// TwinCAT 3 PLC project PLC1
// ProgramVersion: 3.1.4023.0
// libraries:
//   Tc2_EtherCAT, * (Beckhoff Automation GmbH)
//   Tc2_MC2, * (Beckhoff Automation GmbH)
//   Tc2_Standard, * (Beckhoff Automation GmbH)
//   Tc2_SUPS, * (Beckhoff Automation GmbH)
//   Tc2_System, * (Beckhoff Automation GmbH)
//   Tc2_Utilities, * (Beckhoff Automation GmbH)
//   Tc3_MC2_AdvancedHoming, * (Beckhoff Automation GmbH)
//   Tc3_Module, * (Beckhoff Automation GmbH)
//   VisuDialogs, * (System)
// project tree:
//   / GlobalTextList.TcGTLO, PlcTask.TcTTO, Visualization Manager.TcVMO (not stored)
//   GVLs/ GVL_APP.TcGVL
//   POUs/Application_Specific/Applications/ Application_Template.TcPOU
//   POUs/Application_Specific/Axes/ Axis_Template.TcPOU, Pneumatics_Template.TcPOU
//   POUs/ MAIN.TcPOU
//   tc_mca_std_lib/DUTs/Axis_Structures/ ST_AxisConfig.TcDUT, ST_AxisControl.TcDUT, ST_AxisDescription.TcDUT, ST_AxisError.TcDUT, ST_AxisInputs.TcDUT, ST_AxisPersistent.TcDUT, ST_AxisStatus.TcDUT, ST_AxisStruct.TcDUT, ST_GearAxis.TcDUT, ST_HomingConfig.TcDUT
//   tc_mca_std_lib/DUTs/ E_AxisEngUnit.TcDUT, E_AxisParameters.TcTLEO, E_HomingRoutines.TcTLEO, E_MonitoringLedFunction.TcDUT, E_MotionFunctions.TcDUT, E_RestorePosition.TcDUT, E_SlitPairStates.TcDUT, E_SlitPairStatesV2.TcDUT, I_Axis.TcIO, ST_McStatus.TcDUT, ST_MonitoringAlarm.TcDUT
//   tc_mca_std_lib/DUTs/Pneumatics/ E_PneumaticAxisErrors.TcDUT, E_PneumaticMode.TcDUT, ST_PneumaticAxisConfig.TcDUT, ST_PneumaticAxisControl.TcDUT, ST_PneumaticAxisError.TcDUT, ST_PneumaticAxisInputs.TcDUT, ST_PneumaticAxisOutputs.TcDUT, ST_PneumaticAxisStatus.TcDUT, ST_PneumaticAxisStruct.TcDUT
//   tc_mca_std_lib/GVLs/ GVL.TcGVL
//   tc_mca_std_lib/POUs/ FB_ESSMonitoring.TcPOU
//   tc_mca_std_lib/POUs/Motion/ FB_Axis.TcPOU, FB_SlitPair.TcPOU, FB_SlitPairV2.TcPOU
//   tc_mca_std_lib/POUs/Motion/Homing/ FB_Homing.TcPOU
//   tc_mca_std_lib/POUs/Pneumatics/ FB_PneumaticAxis.TcPOU
//   tc_mca_std_lib/VISUs/ languageSupport.TcTLO, MainVisu.TcVIS, ParameterTextList.TcTLO, PneumaticsVisu.TcVIS
//   tc_mca_std_lib/VISUs_Org/ languageSupport_1.TcTLO, MainVisu_1.TcVIS, ParameterTextList_1.TcTLO, PneumaticsVisu_1.TcVIS
// real-time tasks:
//   TASK PlcTask: cycle T#10ms, priority 20, ADS port 350
// motion (NC):
//   TASK NC-Task 1 SAF: cycle T#2ms, priority 4, ADS port 501
//   TASK NC-Task 1 SVB: cycle T#10ms, priority 8, ADS port 511
//   AXIS Axis 1_X1 (id 1)
//     OtherSettings: AllowMotionCmdToSlave=true
//     encoder EncType=1
//     drive DrvType=5
//       Analog: TorqueSetpointScale=10, ScaleFactorActTorque=0.1
//       TimeComp: TaskDelayCycles=1
//     controller CtrType=1
//       CtrPara: PriorControlFactor=1
//         Observer: BandWidth=20
//   AXIS Axis 2_Y (id 2)
//     OtherSettings: AllowMotionCmdToSlave=true
//     encoder EncType=1
//     drive DrvType=5
//       Analog: TorqueSetpointScale=10, ScaleFactorActTorque=0.1
//       TimeComp: TaskDelayCycles=1
//     controller CtrType=1
//       CtrPara: PriorControlFactor=1
//         Observer: BandWidth=20
//   AXIS Axis 3_Z (id 3)
//     OtherSettings: AllowMotionCmdToSlave=true
//     encoder EncType=1
//     drive DrvType=5
//       Analog: TorqueSetpointScale=10, ScaleFactorActTorque=0.1
//       TimeComp: TaskDelayCycles=1
//     controller CtrType=1
//       CtrPara: PriorControlFactor=1
//         Observer: BandWidth=20
//   AXIS Axis 4_X2 (id 4)
//     OtherSettings: AllowMotionCmdToSlave=true
//     encoder EncType=1
//     drive DrvType=5
//       Analog: TorqueSetpointScale=10, ScaleFactorActTorque=0.1
//       TimeComp: TaskDelayCycles=1
//     controller CtrType=1
//       CtrPara: PriorControlFactor=1
//         Observer: BandWidth=20
// variable links:
//   PLC1/PLC1 Instance <-> NC-Task 1 SAF/Axes/Axis 1_X1
//     PlcTask Inputs/GVL.astAxes[1].Axis.NcToPlc <-> Outputs/ToPlc
//     PlcTask Outputs/GVL.astAxes[1].Axis.PlcToNc <-> Inputs/FromPlc
//   PLC1/PLC1 Instance <-> NC-Task 1 SAF/Axes/Axis 2_Y
//     PlcTask Inputs/GVL.astAxes[2].Axis.NcToPlc <-> Outputs/ToPlc
//     PlcTask Outputs/GVL.astAxes[2].Axis.PlcToNc <-> Inputs/FromPlc
//   PLC1/PLC1 Instance <-> NC-Task 1 SAF/Axes/Axis 3_Z
//     PlcTask Inputs/GVL.astAxes[3].Axis.NcToPlc <-> Outputs/ToPlc
//     PlcTask Outputs/GVL.astAxes[3].Axis.PlcToNc <-> Inputs/FromPlc
//   PLC1/PLC1 Instance <-> NC-Task 1 SAF/Axes/Axis 4_X2
//     PlcTask Inputs/GVL.astAxes[4].Axis.NcToPlc <-> Outputs/ToPlc
//     PlcTask Outputs/GVL.astAxes[4].Axis.PlcToNc <-> Inputs/FromPlc

CONFIGURATION PLC1
    RESOURCE PLC ON TwinCAT3
        TASK PlcTask(INTERVAL := T#10ms, PRIORITY := 20);
        PROGRAM MAIN WITH PlcTask : MAIN;
    END_RESOURCE
END_CONFIGURATION

// ---- tc_mca_std_lib/DUTs/Axis_Structures/ST_AxisConfig.TcDUT
(*These are axis parameters that are set up during commissioning and
in theory don't neeed to be change as part of daily moving of axes.
For instance they may be changed due to poor parameter selection
or change of instrument configuration.*)
TYPE ST_AxisConfig :
STRUCT
    //Axis Parameters
    fOverride: LREAL := 100; //Controller override %, used a global scale for an axis in terms of velocity. Generally set to 100%.
    fHomePosition: LREAL := 0; //The position that the axis should be set to once homing is completed
    fHomeFinishDistance: LREAL := 0; //Distrance that the axis should move back into the working zone after homing is finished
    eHomeSeq: E_HomingRoutines; //Homing sequence to perform
    eRestorePosition: E_RestorePosition; //Restore position of incremental axis after loss of power to the CPU, 0=don't restore, 1=restore but don't home

    //Advanced homing parameters
    stHomingConfig: ST_HomingConfig; //Structure containing the advanced homing parameters

    //Temperature disable configuration
    bEnableTemperatureDisable: BOOL := FALSE; //Enable disabling axis because of high temperature
    fMaxTemperature: LREAL := 0.0;
    fTempScalingFactor: REAL := 10.0;

    //Read and Write parameters
    eAxisParameters: E_AxisParameters; //Enumeration of axis parameters
    fWriteAxisParameter: LREAL; //The value to be writen to eAxisParameterNumber
    fReadAxisParameter: LREAL; //Read the current value of the selected eAxisParameterNumber

    //Multi master axis parameters
    astMultiMasterAxis: ARRAY [1..4] OF ST_GearAxis;
    astMultiMasterAxisLatched: ARRAY [1..4] OF ST_GearAxis; //A kind of readback since one doesn't exist in AXIS_REF
    afMultiSlaveAxisRatio: ARRAY [1..GVL_APP.nAXIS_NUM] OF LREAL;

    // Read only MC parameters
    bReadMcParametersValid: BOOL:= FALSE;
    bReadMcParametersError: BOOL:= FALSE;
    fVelocityDefaultSlow: LREAL; //Read only - AxisVeloManSlow
    fVelocityDefaultFast: LREAL; //Read only - AxisVeloManFast
    fHomingVelToCam: LREAL; //Read only - AxisCalibrationVelocityForward
    fHomingVelFromCam: LREAL; //Read only - AxisCalibrationVelocityBackward
    fVeloMax: LREAL; //Read only - AxisMaxVelocity
    fMaxAcc: LREAL; //Read only - AxisMaximumAcceleration
    fMaxDec: LREAL; //Read only - AxisMaxDeceleration
    fDefaultAcc: LREAL; //Read only - AxisDefaultAcceleration
    fDefaultDec: LREAL; //Read only - AxisDefaultDeceleration
    bEnMinSoftPosLimit: BOOL; //Read only
    fMinSoftPosLimit: LREAL; //Read only
    bEnMaxSoftPosLimit: BOOL; //Read only
    fMaxSoftPosLimit: LREAL; //Read only
    bEnPositionLagMonitoring: BOOL; //Read only
    fMaxPosLagValue: LREAL; //Read only
    bEnTargetPositionMonitoring: BOOL; //Read only
    fTargetPositionWindow: LREAL; //Read only
END_STRUCT
END_TYPE

// ---- tc_mca_std_lib/DUTs/Axis_Structures/ST_AxisControl.TcDUT
(*These are parameters that are used to initiate axis movements
They are commands that are commonly used commands*)
TYPE ST_AxisControl :
STRUCT
    //Actions from controls system
    bExecute: BOOL; //Rising edge to execute some motion FB's
    bReset: BOOL; //Reset axis from Error state
    bStop: BOOL;
    bHalt: BOOL;
    bEnable: BOOL; //Enable axis drive
    bJogFwd: BOOL;
    bJogBwd: BOOL;
    bInterlockFwd: BOOL := FALSE; //Bit for interlocking motors in the positive direction
    bInterlockBwd: BOOL := FALSE; //Bit for interlocking motors in the negative direction
    eCommand: E_MotionFunctions;
    fVelocity: LREAL; //Velocity must be specified
    fJogVelocity: LREAL; //Jogging velocity
    fAcceleration: LREAL; //Not all FBs use, 0 is NC default
    fDeceleration: LREAL;
    fPosition: LREAL; //The position to move to for an absolute move and the amount to move in a relative move
    bHWMaskActive: BOOL := FALSE;
    fMaskedTemperature: LREAL := 0.0;
END_STRUCT
END_TYPE

// ---- tc_mca_std_lib/DUTs/Axis_Structures/ST_AxisDescription.TcDUT
TYPE ST_AxisDescription :
STRUCT
    sAxisName : STRING(nMAX_AXIS_NAME);
    eUnit: E_AxisEngUnit; //Code for the axis base unit (like m or degree)
    nPrefix: INT; //Exponent defining unit prefix, e.g. 3 for k(kilo)
END_STRUCT
END_TYPE

// ---- tc_mca_std_lib/DUTs/Axis_Structures/ST_AxisError.TcDUT
TYPE ST_AxisError:
STRUCT
//PLCopen function block errors
    nPowerErrorID: UDINT;
    nMoveAbsoluteErrorID: UDINT;
    nMoveRelativeErrorID: UDINT;
    nMoveVelocityErrorID: UDINT;
    nMoveModuloErrorID: UDINT;
    nHomeErrorID: UDINT;
    nHaltErrorID: UDINT;
    nResetErrorID: UDINT;
    nStopErrorID: UDINT;
    nGearInMultiMasterErrorID: UDINT;
    nGearOutErrorID: UDINT;
    nWriteParameterErrorId: UDINT;
    nReadParameterErrorId: UDINT;
//Error from the NC
    nNCErrorID : UDINT;
END_STRUCT
END_TYPE

// ---- tc_mca_std_lib/DUTs/Axis_Structures/ST_AxisInputs.TcDUT
TYPE ST_AxisInputs :
STRUCT
    bLimitFwd AT %I*: BOOL;
    bLimitBwd AT %I*: BOOL;
    bHomeSensor AT %I*: BOOL; //Reference siganl for homing
    nTempPT100 AT %I*: INT;
END_STRUCT
END_TYPE

// ---- tc_mca_std_lib/DUTs/Axis_Structures/ST_AxisPersistent.TcDUT
TYPE ST_AxisPersistent :
STRUCT
    //Settings for restoring positions on power off
    fPositionAtShutdown: LREAL; //The position that the axis was at when CPU shut down
    fEncoderBiasAtShutdown: LREAL; //Encoder position BIAS value when CPU shut down
    bMovingAtShutdown: BOOL; //True if the axis was moving at shutdown, False otherwise
END_STRUCT
END_TYPE

// ---- tc_mca_std_lib/DUTs/Axis_Structures/ST_AxisStatus.TcDUT
TYPE ST_AxisStatus :
STRUCT
    //Outputs & Status
    bAxisInitialized: BOOL := FALSE; //True when all parameters from actReadMcParameters are valid
    bEnabled: BOOL; //Axis drive enabled
    bCommandAborted: BOOL; //Command aborted output of the eCommand function blocks
    bBusy: BOOL; //Axis busy (eCommand function block is active)
    bDone: BOOL; //Last eCommand function block executed successfully;
    //bDone will also be set with the InGear and InVelocity outputs
    //When InVelocity is set, fbMoveVelocity is still acitve, which is reflected by the bBusy status
    bInVelocity: BOOL; //MC_MoveVelocity has reached target velocity; will stay true until the movement stops
    bHomed: BOOL; //Axis homed
    bMoving: BOOL; //Moving state from the NC
    bMovingForward: BOOL; //Moving forward indicator from NC
    bMovingBackward: BOOL; //Moving backward indicator from NC
    bInTargetPosition: BOOL; //In target position bit from AxisStatus()
    bFwEnabled: BOOL; //Positive movement of axis is enabled/disabled
    bBwEnabled: BOOL; //Negative movement of axis is enabled/disabled
    bInterlockedFwd: BOOL; //Axis interlocked in the postive direction
    bInterlockedBwd: BOOL; //Axis interlocked in the negative direction
    bGeared: BOOL; //Axis is an active slave
    bCoupledGear1: BOOL;
    bCoupledGear2: BOOL;
    bCoupledGear3: BOOL;
    bCoupledGear4: BOOL;
    fActPosition: LREAL; //Actual position value
    fActTemperature: LREAL; //Actual Temperature
    bHighTempAxisDisabled: BOOL := FALSE; //Bit for disabling the axis when temperature too high
    nEncoderRawCounter AT %I*: UDINT; //Raw encoder counter value
    nStepperDriveCounter AT %I*: UDINT; //Raw internal counter from stepper drive
    fActVelocity: LREAL; //Actual velocity
    bError: BOOL; //Motion function block has produced error (NC drive not necessarily in error state)
    nErrorID: UDINT; //Last motion function block errorID or NC errorID
END_STRUCT
END_TYPE

// ---- tc_mca_std_lib/DUTs/Axis_Structures/ST_AxisStruct.TcDUT
TYPE ST_AxisStruct :
STRUCT
    stControl: ST_AxisControl;
    stStatus: ST_AxisStatus;
    stConfig: ST_AxisConfig;
    stError: ST_AxisError;
    stInputs: ST_AxisInputs;
    stDescription: ST_AxisDescription;
    //The NC axis link to the hardware that is controlling
    Axis: AXIS_REF;
END_STRUCT
END_TYPE

// ---- tc_mca_std_lib/DUTs/Axis_Structures/ST_GearAxis.TcDUT
TYPE ST_GearAxis :
STRUCT
    nIndex: UINT := 1; //Index of the master axis
    fRatio: LREAL := 0; //Gearing ratio between master axis and this one
END_STRUCT
END_TYPE

// ---- tc_mca_std_lib/DUTs/Axis_Structures/ST_HomingConfig.TcDUT
TYPE ST_HomingConfig :
STRUCT
    //Hardware signals
    eLimitSwitchMode: MC_Switch_Mode := mcRisingEdge;
    eRefSwitchMode: MC_Switch_Mode := mcRisingEdge;

    //General Advanced Homing Configuration
    bDisableDriveAccess: BOOL := TRUE; //Disables the drive access to drives. Standard for stepper motors. If supported in drive, can be set to FALSE, e.g. for AX5106.
    bEnableLagErrorDetection :BOOL := FALSE; // Keep the lag error detection active during homing
    bInstantLagReduction :BOOL := FALSE; //(belongs to Option4) When referencing to a mechanical fixed stop, it is purposeful in particular with "soft" fixed stops, the lag error is dissipated abruptly by setting this flag.
    tTimeLimit: TIME; // Exceeding this time leads to the search procedure being aborted.
    fDistanceLimit: LREAL; // Exceeding this distance in relation to the start position leads to the search procedure being aborted.
    fTorqueLimit: LREAL; // The motor torque is limited to this value, in relation to the weight counterbalance that is possibly parameterized in the drive, in order to avoid mechanical damage.

    //Homing Configuration for Step Block
    fDetectionVelocityLimit: LREAL; // Velocity that must be fallen below for the DetectionVelocityTime in order to detect driving against the fixed stop.
    tDetectionVelocityTime: TIME; // Time for detecting the velocity undershoot when driving against the fixed stop.
    fLagLimit: LREAL; // Position lag value which, if exceeded, leads to detection of driving against the fixed stop.
END_STRUCT
END_TYPE

// ---- tc_mca_std_lib/DUTs/E_AxisEngUnit.TcDUT
{attribute 'qualified_only'}
{attribute 'strict'}
TYPE E_AxisEngUnit :
(
    eMeter := 0,
    eDegree := 1
) := eMeter;
END_TYPE

// ---- tc_mca_std_lib/DUTs/E_AxisParameters.TcTLEO
{attribute 'qualified_only'}
{attribute 'strict'}
TYPE E_AxisParameters :
(
//PLCopen specific parameters Index-Group 0x4000 + ID
    CommandedPosition := 1, //lreal taken from NcToPlc
    SWLimitForward := 2, //lreal IndexOffset= 16#0001_000E
    SWLimitBackward := 3, //lreal IndexOffset= 16#0001_000D
    EnableLimitForward := 4, //bool IndexOffset= 16#0001_000C
    EnableLimitBackward := 5, //bool IndexOffset= 16#0001_000B
    EnablePositionLagMonitoring := 6, //bool IndexOffset= 16#0002_0010
    MaxPositionLag := 7, //lreal IndexOffset= 16#0002_0012
    AxisMaxVelocity := 8, //lreal IndexOffset= 16#0000_0027
    ActualVelocity := 10, //lreal taken from NcToPlc
    CommandedVelocity := 11, //lreal taken from NcToPlc
    AxisDefaultAcceleration := 12, //lreal IndexOffset= 16#0000_0101
    AxisDefaultDeceleration := 14, //lreal IndexOffset= 16#0000_0102
    AxisDefaultJerk := 16, //lreal IndexOffset= 16#0000_0103

//Beckhoff specific parameters Index-Group 0x4000 + ID
    AxisId := 1000, //lreal IndexOffset= 16#0000_0001
    AxisManualVelocitySlow := 1001, //lreal IndexOffset= 16#0000_0008
    AxisManualVelocityFast := 1002, //lreal IndexOffset= 16#0000_0009
    AxisRapidTraverseVelocity := 1009, //lreal IndexOffset= 16#0000_000A
    AxisVelocityToCam := 1012, //lreal IndexOffset= 16#0000_0006
    AxisVelocityFromCam := 1013, //lreal IndexOffset= 16#0000_0007
    AxisJogIncrementForward := 1014, //lreal IndexOffset= 16#0000_0018
    AxisJogIncrementBackward := 1015, //lreal IndexOffset= 16#0000_0019
    MaxPositionLagFilterTime := 1022, //lreal IndexOffset= 16#0002_0013
    AxisEnPositionRangeMonitoring := 1023, //bool IndexOffset= 16#0000_000F
    AxisPositionRangeWindow := 1024, //lreal IndexOffset= 16#0000_0010
    AxisEnTargetPositionMonitoring:= 1025, //bool IndexOffset= 16#0000_0015
    AxisTargetPositionWindow := 1026, //lreal IndexOffset= 16#0000_0016
    AxisTargetPositionMonitoringTime := 1027, //lreal IndexOffset= 16#0000_0017
    AxisEnInTargetTimeout := 1028, //bool IndexOffset= 16#0000_0029
    AxisInTargetTimeout := 1029, //lreal IndexOffset= 16#0000_002A
    AxisEnMotionMonitoring := 1030, //bool IndexOffset= 16#0000_0011
    AxisMotionMonitoringWindow := 1031, //lreal IndexOffset= 16#0000_0028
    AxisMotionMonitoringTime := 1032, //lreal IndexOffset= 16#0000_0012
    AxisDelayTimeVeloPosition := 1033, //lreal IndexOffset= 16#0000_0104
    AxisEnLoopingDistance := 1034, //bool IndexOffset= 16#0000_0013
    AxisLoopingDistance := 1035, //lreal IndexOffset= 16#0000_0014
    AxisEnBacklashCompensation := 1036, //bool IndexOffset= 16#0000_002B
    AxisBacklash := 1037, //lreal IndexOffset= 16#0000_002C
    AxisEnDataPersistence := 1038, //bool IndexOffset= 16#0000_0030
    AxisRefVeloOnRefOutput := 1039, //lreal IndexOffset= 16#0003_0101
    AxisOverrideType := 1040, //lreal IndexOffset= 16#0000_0105
    //new since 4/2007
    AxisEncoderOffset := 1042, //lreal IndexOffset= 16#0001_0007
    AxisEncoderDirectionInverse := 1043, //bool IndexOffset= 16#0001_0008
    AxisEncoderMask := 1044, //dword IndexOffset= 16#0001_0015
    AxisEncoderModuloValue := 1045, //lreal IndexOffset= 16#0001_0009
    AxisModuloToleranceWindow := 1046, //lreal IndexOffset= 16#0001_001B
    AxisEnablePosCorrection := 1047, //bool IndexOffset= 16#0001_0016
    AxisPosCorrectionFilterTime := 1048, //lreal IndexOffset= 16#0001_0017
    //new since 1/2010
    AxisUnitInterpretation := 1049, //lreal IndexOffset= 16#0000_0026
    AxisMotorDirectionInverse := 1050, //bool  IndexOffset= 16#0003_0006
    //new since 1/2011
    AxisCycleTime := 1051, //lreal IndexOffset= 16#0000_0004
    //new since 5/2011
    AxisFastStopSignalType := 1052, //dword IndexOffset= 16#0000_001E
    AxisFastAcc := 1053, //lreal IndexOffset= 16#0000_010A
    AxisFastDec := 1054, //lreal IndexOffset= 16#0000_010B
    AxisFastJerk := 1055, //lreal IndexOffset= 16#0000_010C
    // new since 1/2012 *)
    AxisEncoderScalingNumerator := 1056, //lreal IndexOffset= 16#0001_0023 - available in Tc3
    AxisEncoderScalingDenominator := 1057, //lreal IndexOffset= 16#0001_0024 - available in Tc3
    (* new since 7/2016 *)
    AxisMaximumAcceleration := 1058, //lreal IndexOffset= 16#0000_00F1
    AxisMaximumDeceleration := 1059, //lreal IndexOffset= 16#0000_00F2
    AxisVeloJumpFactor := 1060, //lreal IndexOffset= 16#0000_0106
    AxisToleranceBallAuxAxis := 1061, //lreal IndexOffset= 16#0000_0108
    AxisMaxPositionDeviationAuxAxis := 1062, //lreal IndexOffset= 16#0000_0109
    AxisErrorPropagationMode := 1063, //dword IndexOffset= 16#0000_001A
    AxisErrorPropagationDelay := 1064, //lreal IndexOffset= 16#0000_001B
    AxisCoupleSlaveToActualValues := 1065, //bool IndexOffset= 16#0000_001C
    AxisAllowMotionCmdToSlaveAxis := 1066, //bool IndexOffset= 16#0000_0020
    AxisAllowMotionCmdToExtSetAxis := 1067, //bool IndexOffset= 16#0000_0021
    AxisEncoderSubMask := 1068, //dword IndexOffset= 16#0001_0108
    AxisEncoderReferenceSystem := 1069, //dword IndexOffset= 16#0001_0019
    AxisEncoderPositionFilterPT1 := 1070, //lreal IndexOffset= 16#0001_0010
    AxisEncoderVelocityFilterPT1 := 1071, //lreal IndexOffset= 16#0001_0011
    AxisEncoderAccelerationFilterPT1 := 1072, //lreal IndexOffset= 16#0001_0012
    AxisEncoderMode := 1073, //dword IndexOffset= 16#0001_000A
    AxisEncoderHomingInvDirCamSearch := 1074, //bool IndexOffset= 16#0001_0101
    AxisEncoderHomingInvDirSyncSearch := 1075, //bool IndexOffset= 16#0001_0102
    AxisEncoderHomingCalibValue := 1076, //lreal IndexOffset= 16#0001_0103
    AxisEncoderReferenceMode := 1077, //dword IndexOffset= 16#0001_0107
    AxisRefVeloOutputRatio := 1078, //lreal IndexOffset= 16#0003_0102
    AxisDrivePositionOutputScaling := 1079, //lreal IndexOffset= 16#0003_0109
    AxisDriveVelocityOutputScaling := 1080, //lreal IndexOffset= 16#0003_0105
    AxisDriveVelocityOutputDelay := 1081, //lreal IndexOffset= 16#0003_010D
    AxisDriveMinOutputLimitation := 1082, //lreal IndexOffset= 16#0003_000B
    AxisDriveMaxOutputLimitation := 1083, //lreal IndexOffset= 16#0003_000C
    AxisTorqueInputScaling := 1084, //lreal IndexOffset= 16#0003_0031 - available in Tc3
    AxisTorqueInputFilterPT1 := 1085, //lreal IndexOffset= 16#0003_0032 - available in Tc3
    AxisTorqueDerivationInputFilterPT1 := 1086, //lreal IndexOffset= 16#0003_0033 - available in Tc3
    AxisTorqueOutputScaling := 1087, //lreal IndexOffset= 16#0003_010B
    AxisTorqueOutputDelay := 1088, //lreal IndexOffset= 16#0003_010F
    AxisAccelerationOutputScaling := 1089, //lreal IndexOffset= 16#0003_010A
    AxisAccelerationOutputDelay := 1090, //lreal IndexOffset= 16#0003_010E
    AxisDrivePositionOutputSmoothFilterType := 1091, //dword IndexOffset= 16#0003_0110
    AxisDrivePositionOutputSmoothFilterTime := 1092, //lreal IndexOffset= 16#0003_0111
    AxisDrivePositionOutputSmoothFilterOrder := 1093, //dword IndexOffset= 16#0003_0112
    AxisDriveMode := 1094, //dword IndexOffset= 16#0003_000A
    AxisDriftCompensationOffset := 1095, //lreal IndexOffset= 16#0003_0104
    AxisPositionControlKv := 1096, //lreal IndexOffset= 16#0002_0102
    AxisCtrlVelocityPreCtrlWeight := 1097, //lreal IndexOffset= 16#0002_000B
    AxisControllerMode := 1098, //dword IndexOffset= 16#0002_000A
    AxisCtrlAutoOffset := 1099, //bool IndexOffset= 16#0002_0110
    AxisCtrlAutoOffsetTimer := 1100, //lreal IndexOffset= 16#0002_0115
    AxisCtrlAutoOffsetLimit := 1101, //lreal IndexOffset= 16#0002_0114
    AxisSlaveCouplingControlKcp := 1102, //lreal IndexOffset= 16#0002_010F
    AxisCtrlOutputLimit := 1103, //lreal IndexOffset= 16#0002_0100

//Beckhoff specific axis status information - READ ONLY Index-Group 0x4100 + ID
    AxisTargetPosition := 2000, //lreal IndexOffset= 16#0000_0013
    AxisRemainingTimeToGo := 2001, //lreal IndexOffset= 16#0000_0014
    AxisRemainingDistanceToGo := 2002, //lreal IndexOffset= 16#0000_0022, 16#0000_0042

//Beckhoff specific axis functions
    //read/write gear ratio of a slave
    AxisGearRatio := 3000, //lreal read: IndexGroup=0x4100+ID, IdxOffset=16#0000_0022,
                                 //write:IndexGroup=0x4200+ID, IdxOffset=16#0000_0042

//Beckhoff specific other parameters
    //new since 1/2011
    NcSafCycleTime := 4000, //lreal IndexOffset= 16#0000_0010
    NcSvbCycleTime := 4001 //lreal IndexOffset= 16#0000_0012

);
END_TYPE

// ---- tc_mca_std_lib/DUTs/E_HomingRoutines.TcTLEO
{attribute 'qualified_only'}
{attribute 'strict'}
TYPE E_HomingRoutines :
(
    eNoHoming := 0,

    //0X: LIMIT Switch
    //Home to bBwdLimit, record position on first approach
    eHomeToLimit_Bwd := 1,
    //Home to bFwdLimit, record position on first approach
    eHomeToLimit_Fwd := 2,
    //Find bBwdLimit (using towardsCam speed), then reverse direction looking FOR falling edge (using fromCam speed)
    //eHomeToLimit_Bwd_2Speeds := 3,
    //Find bFwdLimit (using towardsCam speed), then reverse direction looking for falling edge (using fromCam speed)
    //eHomeToLimit_Fwd_2Speeds := 4,

    //1X: Home Sensor
    //Home to bHome in Bwd direction (will reverse direction if limit hit), record position on first approach
    eHomeToRef_Bwd := 11,
    //Home to bHome in Fwd direction (will reverse direction if limit hit), record position on first approach
    eHomeToRef_Fwd := 12,
    //Find bHome in Bwd direction (using towardsCam speed) then reverse direction looking for falling edge (using fromCam speed), will reverse direction if limit hit
    //eHomeToRef_Bwd_2Speeds := 13,
    //Find bHome in Fwd direction (using towardsCam speed) then reverse direction looking for falling edge (using fromCam speed), will reverse direction if limit hit
    //eHomeToRef_Fwd_2Speeds := 14,

    //2X: Enc Pulse
    //Home to EncRefPulse in Bwd direction (used for single turn rotary axis without limit switches)
    eHomeToEncPulse_Bwd := 21,
    //Home to EncRefPulse in Fwd direction (used for single turn rotary axis without limit switches)
    eHomeToEncPulse_Fwd := 22,
    //Home to EncRefPulse via bBwdLimit (using towardsCam speed), then reverse direction looking for falling edge on ref pulse (using fromCam speed)
    eHomeToEncPulse_viaBwdLimit := 23,
    //Home to EncRefPulse via bFwdLimit (using towardsCam speed), then reverse direction looking for falling edge on ref pulse (using fromCam speed)
    eHomeToEncPulse_viaFwdLimit := 24,

    //3X: Home To Mechanical Block (Lag based StepBlockDetection)
    //Home towards a mechanical block in Bwd direction
    eHomeToBlock_Bwd := 30,
    //Home towards a mechanical block in Fwd direction
    eHomeToBlock_Fwd := 31,

    //9X: Software
    eHomeDirect := 90 //Set position directly to fHomePosition
) := eHomeDirect;
END_TYPE

// ---- tc_mca_std_lib/DUTs/E_MonitoringLedFunction.TcDUT

{attribute 'qualified_only'}
{attribute 'strict'}
TYPE E_MonitoringLedFunction :
(
    eUndefined := 0,
    eSteady := 1,
    eSlow := 2,
    eFast := 3
);
END_TYPE

// ---- tc_mca_std_lib/DUTs/E_MotionFunctions.TcDUT
{attribute 'qualified_only'}
{attribute 'strict'}
TYPE E_MotionFunctions :
(
    eMoveAbsolute := 0,
    eMoveRelative := 1,
    eMoveVelocity := 2, //Continous moving at a set velocity once bExecute goes high
    eMoveModulo := 3, //Move for 360 deg rotation, see Beckhoff docs
    eGearInMultiMaster := 4, //Gears in this axis to be the slave of the axis specified in stMultiMasterAxis with the ratio specified
    eGearOut := 5, //Removes gearing set in the above command
    eHome := 10, //Run the homing routine for the axis
    eWriteParameter := 50, //Writes the set value to the set parameter once bExecute goes high
    eReadParameter := 60 //Reads a single Parameter
) := eHome; //Home is the default behaviour of the axis.
END_TYPE

// ---- tc_mca_std_lib/DUTs/E_RestorePosition.TcDUT
{attribute 'qualified_only'}
{attribute 'strict'}
TYPE E_RestorePosition :
(
    eDontRestore :=0,
    eRestoreWithoutHome := 1 //Redefined the position of the axis to that when the power was lost
);
END_TYPE

// ---- tc_mca_std_lib/DUTs/E_SlitPairStates.TcDUT
{attribute 'qualified_only'}
{attribute 'strict'}
TYPE E_SlitPairStates :
(
    INIT := 0,
    INIT_CLEAR_GEARING,
    INIT_GEAROUT_CHECK,
    CHECK_HOME_STATUS,
    HOME_BLADES,
    CHECK_BLADE_HOME_COMPLETE,
    HOME_GAP,
    CHECK_GAP_HOME_COMPLETE,
    GEARIN_SLITS,
    CHECK_GEARIN_SLITS_COMPLETE,
    SLITS_OPERATIONAL,
    GEAROUT_BLADES,
    CHECK_GEAROUT_COMPLETE,
    CLEAR_GAP_CALIBRATION,
    ERROR,
    ERROR_GEAROUT,
    ERROR_GEAROUT_CHECK,
    ERROR_RESET_AXES,
    ERROR_RESET_CHECK
);
END_TYPE

// ---- tc_mca_std_lib/DUTs/E_SlitPairStatesV2.TcDUT

{attribute 'qualified_only'}
{attribute 'strict'}
TYPE E_SlitPairStatesV2 :
(
    eInit := 0,
    eEnableRealGenerators,
    eDisableRealGenerators,
    eEnableVirtualGenerators,
    eDisableVirtualGenerators,
    eWaitForVirtualMoveDone,
    eWaitForRealMoveDone,
    eError,
    eOperational,
    eWaitForVirtualHomed,
    eWaitForRealHomed,
    eCheckRealAxisGeneratorsEnabled,
    eCheckVirtualAxisGeneratorsEnabled
);
END_TYPE

// ---- tc_mca_std_lib/DUTs/Pneumatics/E_PneumaticAxisErrors.TcDUT
{attribute 'qualified_only'}
{attribute 'strict'}
TYPE E_PneumaticAxisErrors :
(
    eNoError := 0,
    eExtractTimedOut := 1, //Extraction movement not done in expected time
    eRetractTimedOut := 2, //Retraction movement not done in expected time
    eNotMovingExtract := 3, //Extract command not executed, cylinder stays in place
    eNotMovingRetract := 4, //Retract command not executed, cylinder stays in place
    eInterlockOn := 5, //Interlock signal on, cylinder retracts to Limit Bwd
    eNoPSSPermit := 6, //Permit signal lost, cylinder retracts to Limit Bwd
    eAirPressureError := 7 //Air pressure signal out of range
):= eNoError;
END_TYPE

// ---- tc_mca_std_lib/DUTs/Pneumatics/E_PneumaticMode.TcDUT
{attribute 'qualified_only'}
{attribute 'strict'}
TYPE E_PneumaticMode :
(   eSingleSolenoidControl := 0, //Single solenoid valve with spring return
    eReset := 1,
    eError := 2
):= eSingleSolenoidControl;
END_TYPE

// ---- tc_mca_std_lib/DUTs/Pneumatics/ST_PneumaticAxisConfig.TcDUT
TYPE ST_PneumaticAxisConfig :
STRUCT
    nTimeToExtend: INT; //User defined time for the cylider to extract in seconds
    nTimeToRetract: INT; //User defined time for the cylinder to retract in seconds
END_STRUCT
END_TYPE

// ---- tc_mca_std_lib/DUTs/Pneumatics/ST_PneumaticAxisControl.TcDUT
TYPE ST_PneumaticAxisControl :
STRUCT
    bExtend: BOOL; //Variable to control solenoid valve from PLC
    bRetract: BOOL; //Variable to control solenoid valve from PLC
    bInterlock: BOOL; //Input interlock signal for the movement
    bReset: BOOL; //Reset signal from EPICS
END_STRUCT
END_TYPE

// ---- tc_mca_std_lib/DUTs/Pneumatics/ST_PneumaticAxisError.TcDUT
TYPE ST_PneumaticAxisError :
STRUCT
    bExtendCylinderTimedOut : BOOL; //Pneumatic cylinder didn't extend in givne time
    bRetractCylinderTimedOut : BOOL; //Pneumatic cylinder didn't retract in given time
    bNoPermit : BOOL; //No permit to move the cylinder
END_STRUCT
END_TYPE

// ---- tc_mca_std_lib/DUTs/Pneumatics/ST_PneumaticAxisInputs.TcDUT
TYPE ST_PneumaticAxisInputs :
STRUCT
    bEndSwitchFwd AT %I*: BOOL; //End Switch Fwd input
    bEndSwitchBwd AT %I*: BOOL; //End Switch Bwd input
    bSolenoidActive AT %I*: BOOL; //Solenoid valve Extend Input (for single solenoid)
    bPSSPermit AT %I*: BOOL; //Input signal from PSS for the movement
    bPressureExtend AT %I*: BOOL; //Input signal of air pressure for cyclinder extraction
    bPressureRetract AT %I*: BOOL; //Input signal of air pressure for cylinder retraction
    nAirPressureValve AT %I*: REAL; //Input signal of air pressure for pneumatic valve
    bOpenManual AT %I*: BOOL; //Push button input to extend cylinder
    bCloseManual AT %I*: BOOL; //Push button input to retract the cylinder
END_STRUCT
END_TYPE

// ---- tc_mca_std_lib/DUTs/Pneumatics/ST_PneumaticAxisOutputs.TcDUT
TYPE ST_PneumaticAxisOutputs :
STRUCT
    bEndSwitchFwdOn AT %Q*: BOOL; //End Switch Fwd power output
    bEndSwitchBwdOn AT %Q*: BOOL; //End Switch Bwd power output
    bValveOn AT %Q*: BOOL; //Output of the solenoid valve (for single solenoid)
    bPressureExtendOn AT %Q*: BOOL; //Power output for air pressure switch
    bPressureRetractOn AT %Q*: BOOL; //Power output for air pressure switch
    fAirPressureOn AT %Q*: REAL; //Power output for analog pressure sensor
END_STRUCT
END_TYPE

// ---- tc_mca_std_lib/DUTs/Pneumatics/ST_PneumaticAxisStatus.TcDUT
TYPE ST_PneumaticAxisStatus :
STRUCT
    bExtending: BOOL; //Extending movement status
    bRetracting: BOOL; //Retraction movement status
    bExtended: BOOL; //Cylinder extracted status
    bRetracted: BOOL; //Cylinder retracted status
    nTimeElapsedExtend: INT; //Elapsed time while extracting cylinder
    nTimeElapsedRetract: INT; //Elapsed time while retracting cylinder
    bSolenoidActive: BOOL; //Status input of valve solenoid
    sStatus: STRING; //Pneumatic cylinder current status
    bInterlocked: BOOL; //Interlock siganl active
    bPSSPermitOK: BOOL; //Status of the PSS permit signal
    bError: BOOL; //Pneumatic axis is in Error state
END_STRUCT
END_TYPE

// ---- tc_mca_std_lib/DUTs/Pneumatics/ST_PneumaticAxisStruct.TcDUT
TYPE ST_PneumaticAxisStruct :
STRUCT
    stPneumaticAxisInputs: ST_PneumaticAxisInputs;
    stPneumaticAxisOutputs: ST_PneumaticAxisOutputs;
    stPneumaticAxisControl: ST_PneumaticAxisControl;
    stPneumaticAxisStatus: ST_PneumaticAxisStatus;
    stPneumaticAxisConfig: ST_PneumaticAxisConfig;
    ePneumaticAxisMode: E_PneumaticMode;
    ePneumaticAxisErrors: E_PneumaticAxisErrors;
END_STRUCT
END_TYPE

// ---- tc_mca_std_lib/DUTs/ST_McStatus.TcDUT
TYPE ST_McStatus :
STRUCT
    Done: BOOL;
    Busy: BOOL;
    Active: BOOL;
    InVelocity: BOOL;
    CommandAborted: BOOL;
    Error: BOOL;
    ErrorID: UDINT;
END_STRUCT
END_TYPE

// ---- tc_mca_std_lib/DUTs/ST_MonitoringAlarm.TcDUT

TYPE ST_MonitoringAlarm :
STRUCT
    bAlarmSet: BOOL;
    bAlarmReset: BOOL;
    nStatusLED: E_MonitoringLedFunction;
    nWarningLED: E_MonitoringLedFunction;
    nEmergencyLED: E_MonitoringLedFunction;
    nAcknowledgeLED: E_MonitoringLedFunction;
    nErrorID: INT;
    sErrorMsg: STRING;
    bAlarmActive: BOOL;
END_STRUCT
END_TYPE

// ---- GVLs/GVL_APP.TcGVL
{attribute 'qualified_only'}
VAR_GLOBAL
END_VAR

VAR_GLOBAL CONSTANT
    nAXIS_NUM: UINT := 4;
	nPNEUMATIC_AXIS_NUM:  UINT := 2;
END_VAR

// ---- tc_mca_std_lib/GVLs/GVL.TcGVL
VAR_GLOBAL
    // Semantic version in machine-readable format.
    // Update it and commit it immediatly before setting a tag
    nVersionMajor: UINT := 2; // Major Version
    nVersionMinor: UINT := 2; // Minor Version
    nVersionPatch: UINT := 0; // Patch level
    astAxes: ARRAY [1..GVL_APP.nAXIS_NUM] OF ST_AxisStruct; //Array of ST_AxisStruct for holding axis parameters and controls
    astPneumaticAxes: ARRAY [1..GVL_APP.nPNEUMATIC_AXIS_NUM] OF ST_PneumaticAxisStruct; //Array of ST_PneumaticAxisStruct for holding pneumatic axis parameters and controls
    iAxis: UINT; //Index for for loops while going through axes
    iPneumaticAxis: UINT := 1; //Index for for loops while going through pneumatic axes
    fbGetCurTaskIndex: GETCURTASKINDEX;
    bLocalMode: BOOL;
END_VAR

VAR_GLOBAL CONSTANT
    nMAX_AXIS_NAME: UINT := 32;
END_VAR

VAR_GLOBAL PERSISTENT
    astAxesPersistent: ARRAY [1..GVL_APP.nAXIS_NUM] OF ST_AxisPersistent;
END_VAR

// ---- tc_mca_std_lib/DUTs/I_Axis.TcIO
INTERFACE I_Axis

METHOD EndOfCycle : BOOL
VAR_INPUT
END_VAR
END_METHOD

METHOD Run : BOOL
VAR_INPUT
END_VAR
END_METHOD

PROPERTY stAxis : REFERENCE TO ST_AxisStruct
GET
END_GET
SET
END_SET
END_PROPERTY

END_INTERFACE

// ---- POUs/MAIN.TcPOU
PROGRAM MAIN
VAR
    sVersion: STRING := '1.0.0';
    aIAxes: ARRAY [1..GVL_APP.nAXIS_NUM] OF I_Axis;
    afbAxes: ARRAY [1..GVL_APP.nAXIS_NUM] OF FB_Axis;
    afbPneumaticAxes: ARRAY [1..GVL_APP.nPNEUMATIC_AXIS_NUM] OF FB_PneumaticAxis;
    hmiAxisSelection: INT := 1; //Not possible to use local hmi variables for array indexes
    hmiPneumaticAxisSelection: INT := 1;
//Startup, Shutdown and UPS
    fbUPS: FB_S_UPS_CX51x0;
    eUpsMode: E_S_UPS_Mode := eSUPS_WrPersistData_Shutdown;
    eStartUp: (eColdStart, eReadAxisFeedbackType, eCheckReadDone, eExecuteRestore, eCheckRestore, eFinishRestore);
    bPositionRestoreDone: BOOL := FALSE;
    bRestoreExecute: BOOL := FALSE;
    bExecuteReadEncRefSys: BOOL := FALSE;
    nRetry: INT;
    iAxes: UINT; //index for for loops in Position recovery actions
    afbReadEncRefSys: ARRAY [1..GVL_APP.nAXIS_NUM] OF MC_ReadParameter;
    afbSetPosition: ARRAY [1..GVL_APP.nAXIS_NUM] OF MC_SetPosition;
    afbReadPositionBias: ARRAY [1..GVL_APP.nAXIS_NUM] OF MC_ReadParameter;
    afbWritePositionBias: ARRAY [1..GVL_APP.nAXIS_NUM] OF MC_WriteParameter;
    fbGetDeviceIdentification: FB_GetDeviceIdentificationEx;
END_VAR

VAR PERSISTENT
    bRestoreOnStartup: BOOL;
END_VAR

POSITION_RECOVERY();
PROG();
AXES();

ACTION AXES:
//First cycle, assign FB_axis to interface array
IF _TaskInfo[fbGetCurTaskIndex.index].FirstCycle THEN
    FOR GVL.iAxis := 1 TO GVL_APP.nAXIS_NUM DO
        afbAxes[GVL.iAxis].stAxis REF= astAxes[GVL.iAxis];
        aIAxes[GVL.iAxis] := afbAxes[GVL.iAxis];
    END_FOR
    //Custom axis types defined and linked to aiAxes here
      //FB_CustomAxis extends FB_axis
        //fbCustomAxis.stAxis REF= astAxes[x];
        //aIAxes[x] := fbCustomAxis;
END_IF

//Execute FB_Axis logic
FOR GVL.iAxis := 1 TO GVL_APP.nAXIS_NUM DO
    aIAxes[GVL.iAxis].Run();
END_FOR

//Execute Pneumatic Axis logic
FOR GVL.iPneumaticAxis := 1 TO GVL_APP.nPNEUMATIC_AXIS_NUM DO
    afbPneumaticAxes[GVL.iPneumaticAxis](stPneumaticAxisStruct := GVL.astPneumaticAxes[GVL.iPneumaticAxis]);
END_FOR
END_ACTION

ACTION CHECK_UPS:
fbUPS(eUpsMode := eUpsMode);

FOR iAxes := 1 TO GVL_APP.nAXIS_NUM DO
    //Read encoder position BIAS
    IF astAxes[iAxes].stStatus.bAxisInitialized THEN
        afbReadPositionBias[iAxes](Axis := GVL.astAxes[iAxes].Axis,
                        Enable := TRUE,
                        ReadMode:= READMODE_CYCLIC,
                        ParameterNumber := E_AxisParameters.AxisEncoderOffset);
    END_IF
END_FOR

IF eGlobalSUpsState = eSUPS_PowerFailure THEN
    //first cycle of powerfailure
    //execute code that should only be done once with each powerfailure, i.e. increase powerfailure counter
    bRestoreOnStartup := TRUE;
    STORE_PERSISTENT();
    RETURN;
ELSIF eGlobalSUpsState <> eSUPS_PowerOK THEN
    //next cycles of powerfailure
    //skip regular code execution for the remaining cycles of the powerfailure/writing of persistent data/quick shutdown...
    RETURN;
END_IF
END_ACTION

ACTION POSITION_RECOVERY:
fbGetDeviceIdentification(bExecute := TRUE);
IF (fbGetDeviceIdentification.stDevIdent.strHardwareSerialNo <> '') THEN
    CHECK_UPS();
    RESTORE_POSITIONS();
END_IF
END_ACTION

ACTION PROG:
//Get task index for Axes parameters initialization.
GVL.fbGetCurTaskIndex();

//Call the programs that are defined in the "Application Specific" folder.
//Create as many programs in that folder as axes and applications you have or need

//Axes initial parameters and program
Axis_Template();
//Pneumatics_Template();

//Application program calls
Application_Template();
END_ACTION

ACTION RESTORE_POSITIONS:
//This ACT will restore the position of an incremental axis on startup with the act position it read before losing power.
//It checks the type of axis, 0=incremental, and that the axis was stationary at shut down.
//Because 0 equates to incremental we also need to check that the data is valid, otherwise by default it would restore all axes.
//By default an axis will not restore the position unless it is set to opt-in, i.e. GVL.aAxes[iAxes].stConfig.eRestorePosition is non-zero.
//This needs to be initialised somewhere in TwinCAT code otherwise it will not be available at start up.
//A restore will only be performed on a loss of power, this code shouldn't make any changes on a reset cold, a rest origin or a download.
//There is a enum to allow for different types of restore modes, currently only one is implemented.
//0 'DontRestore'
//1 'RestoreWithoutHome' -restores the position using a set position fb and does not set the home bit in the axis struct.
//Note from Beckhoff: "A maximum of 1 MB persistent data can be reliably saved over the entire service life."
//Encoder Reference system types: https://infosys.beckhoff.com/english.php?content=../content/1033/tf50x0_tc3_nc_ptp/3439907723.html&id=
//INCREMENTAL=0;
//ABSOLUTE=1;
//ABSOLUTE (modulo)=2;
//ABSOLUTE MULTITURN RANGE (with single overflow)=3;
//INCREMENTAL (singleturn absolute)=4;
//ABSOLUTE SINGLETURN RANGE (with single overflow)=5;


IF bRestoreOnStartup AND eGlobalSUpsState = eSUPS_PowerOK THEN
    bRestoreOnStartup := FALSE;
    bRestoreExecute := TRUE;
END_IF

//Upon startup bPositionRestoreDone will be set to FALSE, after successfully completing the following code it will be set TRUE
//and should stay TRUE for the rest of the time the PLC is operational, thus this routine should only be completed once.
IF bRestoreExecute AND NOT bPositionRestoreDone THEN
    //Cycle through function blocks that read the encoder reference system i.e. whether axis is incremental or absolute
    FOR iAxes := 1 TO GVL_APP.nAXIS_NUM DO
         afbReadEncRefSys[iAxes](
            Axis := GVL.astAxes[iAxes].Axis,
            ParameterNumber := MC_AxisParameter.AxisEncoderReferenceSystem,
            ReadMode := E_READMODE.READMODE_ONCE);
    END_FOR

    //Cycle through set position and MC_WritePArameter function blocks for each axis
    FOR iAxes := 1 TO GVL_APP.nAXIS_NUM DO
        afbSetPosition[iAxes](
            Axis := GVL.astAxes[iAxes].Axis,
            Position := astAxesPersistent[iAxes].fPositionAtShutdown);

        afbWritePositionBias[iAxes](
            Axis:= GVL.astAxes[iAxes].Axis,
            ParameterNumber:= E_AxisParameters.AxisEncoderOffset,
            Value:= astAxesPersistent[iAxes].fEncoderBiasAtShutdown);
    END_FOR

    CASE eStartUp OF
        eColdStart:
            //First cycle of the PLC, do nothing just give one cycle for variables to initialise
            IF NOT bPositionRestoreDone THEN
                eStartUp := eReadAxisFeedbackType;
                nRetry := 0;
            END_IF

        eReadAxisFeedbackType:
            //Exectute the function blocks to read the encoder reference system (0=inc OR 1=ABS)
            FOR iAxes := 1 TO GVL_APP.nAXIS_NUM DO
                afbReadEncRefSys[iAxes].Enable := TRUE;
                eStartUp := eCheckReadDone;
            END_FOR

        eCheckReadDone:
            //Check the encoder reference system has been read for all axis -> if busy then continue with PLC cycle and check again next time.
            //If afbReadEncRefSys not started then go back a step.
            //If any axes result in an error the code will get stuck here, this happens if GVL_APP.nAXIS_NUM is not set correctly
            FOR iAxes := 1 TO GVL_APP.nAXIS_NUM DO
                IF NOT afbReadEncRefSys[iAxes].Valid THEN
                    IF afbReadEncRefSys[iAxes].Busy THEN
                        //Exit MAIN.STARTUP Action and wait till next cycle, needs to cycle through whole program in order for data to update
                        RETURN;
                    ELSE
                        //Sometimes the code gets here and the afbReadEncRefSys[iAxes] misses the rising edge. If  the code gets here it means
                        //valid=FALSE and .busy=FALSE which indicateds the FB probably hasn't started and thus needs to see a rising edge.
                        //Set execute to low, Exit MAIN.STARTUP and go back a step in the CASE statement.
                        afbReadEncRefSys[iAxes].Enable := FALSE;
                        eStartUp := eReadAxisFeedbackType;
                        nRetry := nRetry + 1; //counter used for troubleshooting to see how many cycles it takes before afbReadEncRefSys function blocks are read correctly
                        RETURN;
                    END_IF
                END_IF
            END_FOR
            //If the code gets here all axes have .valid=TRUE for all axes
            eStartUp := eExecuteRestore;

        eExecuteRestore:
            //Execute position and encoder BIAS restore by setting Execute = TRUE
           FOR iAxes := 1 TO GVL_APP.nAXIS_NUM DO
                IF GVL.astAxes[iAxes].stConfig.eRestorePosition = E_RestorePosition.eRestoreWithoutHome THEN
                    //Restore position value for incremental encoders
                    IF NOT astAxesPersistent[iAxes].bMovingAtShutdown AND
                    (afbReadEncRefSys[iAxes].Value = 0 OR
                     afbReadEncRefSys[iAxes].Value = 2 OR
                     afbReadEncRefSys[iAxes].Value = 4) THEN
                       afbSetPosition[iAxes].Execute := TRUE;
                    //Restore encoder position BIAS for absolute encoders
                    ELSIF afbReadEncRefSys[iAxes].Value = 1 OR
                    afbReadEncRefSys[iAxes].Value = 3 OR
                    afbReadEncRefSys[iAxes].Value = 5 THEN
                       afbWritePositionBias[iAxes].Execute := TRUE;
                    END_IF
                ELSE
                    RETURN;
                END_IF
            END_FOR
            eStartUp := eCheckRestore;


        eCheckRestore:
            //Check the set position and write enocder BIAS fbs are finished
            //Nothing actually happens if the restore is not done, the code just returns from here each cycle and the
            //bPositionRestoreDone will never get set to TRUE and will take up cycle time
            FOR iAxes := 1 TO GVL_APP.nAXIS_NUM DO
                IF GVL.astAxes[iAxes].stConfig.eRestorePosition = E_RestorePosition.eRestoreWithoutHome THEN
                    IF NOT astAxesPersistent[iAxes].bMovingAtShutdown AND
                    (afbReadEncRefSys[iAxes].Value = 0 OR
                     afbReadEncRefSys[iAxes].Value = 2 OR
                     afbReadEncRefSys[iAxes].Value = 4) THEN
                        IF NOT afbSetPosition[iAxes].Done THEN
                            afbSetPosition[iAxes].Execute := FALSE;
                            eStartUp := eExecuteRestore;
                            RETURN;
                        END_IF
                     ELSIF afbReadEncRefSys[iAxes].Value = 1 OR
                     afbReadEncRefSys[iAxes].Value = 3 OR
                     afbReadEncRefSys[iAxes].Value = 5 THEN
                        IF NOT afbWritePositionBias[iAxes].Done THEN
                            afbWritePositionBias[iAxes].Execute := FALSE;
                            eStartUp := eExecuteRestore;
                            RETURN;
                        END_IF
                    END_IF
                ELSE
                    RETURN;
                END_IF
            END_FOR
            eStartUp :=  eFinishRestore;

        eFinishRestore:
            //Remove execute = TRUE for afbRestorePosition and fbWritePositionBias
            FOR iAxes := 1 TO GVL_APP.nAXIS_NUM DO
                afbSetPosition[iAxes].Execute := FALSE;
                afbWritePositionBias[iAxes].Execute := FALSE;
                bPositionRestoreDone := TRUE;
                bRestoreExecute := FALSE;
            END_FOR
    END_CASE
END_IF
END_ACTION

ACTION STORE_PERSISTENT:
FOR iAxes := 1 TO GVL_APP.nAXIS_NUM DO
    //Store Position beofre shutdown
    astAxesPersistent[iAxes].fPositionAtShutdown := GVL.astAxes[iAxes].Axis.NcToPlc.ActPos;

    //Store encoder position BIAS at shutdown
    astAxesPersistent[iAxes].fEncoderBiasAtShutdown := afbReadPositionBias[iAxes].Value;

    //Store value of moving at shutdown
    IF GVL.astAxes[iAxes].Axis.Status.StandStill OR GVL.astAxes[iAxes].Axis.Status.Disabled THEN
        astAxesPersistent[iAxes].bMovingAtShutdown := FALSE;
    ELSE
        astAxesPersistent[iAxes].bMovingAtShutdown := TRUE;
    END_IF
END_FOR
END_ACTION

END_PROGRAM

// ---- tc_mca_std_lib/POUs/Motion/FB_Axis.TcPOU
//Function block to run a virtual drive with Nc
FUNCTION_BLOCK FB_Axis IMPLEMENTS I_axis
VAR
    _stAxis: REFERENCE TO ST_AxisStruct; // Local property pointer for axis structure
    astMcStatus: ARRAY[1..nMCSTATUS_ARRAY_SIZE] OF POINTER TO ST_McStatus; //Array of all MC status signals defined in FB_init

    fbPower: MC_Power;
    stMcStatusPower: ST_McStatus;

    fbStop: MC_Stop;
    stMcStatusStop: ST_McStatus;

    fbHalt: MC_Halt;
    stMcStatusHalt: ST_McStatus;

    fbReset: MC_Reset;
    stMcStatusReset: ST_McStatus;

    fbMoveAbsolute: MC_MoveAbsolute;
    fbMoveAbsolute2: MC_MoveAbsolute;
    stMcStatusMoveAbsolute: ST_McStatus;

    fbMoveRelative: MC_MoveRelative;
    stMcStatusMoveRelative: ST_McStatus;

    fbMoveVelocity: MC_MoveVelocity;
    stMcStatusMoveVelocity: ST_McStatus;

    fbMoveModulo: MC_MoveModulo;
    fbMoveModulo2: MC_MoveModulo;
    stMcStatusMoveModulo: ST_McStatus;

    fbHome: FB_Homing;
    stMcStatusHome: ST_McStatus;

    fbReadParameter: MC_ReadParameter;
    stMcStatusReadParameter: ST_McStatus;

    fbWriteParameter: MC_WriteParameter;
    stMcStatusWriteParameter: ST_McStatus;

    fbGearIn: MC_GearIn;
    stMcStatusGearIn: ST_McStatus;

    fbGearOut: MC_GearOut;
    stMcStatusGearOut: ST_McStatus;

    stMasterAxis: ST_GearAxis := (nIndex := 1, fRatio := 0);
    nSlaveAxesIndex: UINT;
    nAxisIndex: UINT;
    nMultiMastersAxesIndex: UINT;

    fbGearInMultiMaster: MC_GearInMultiMaster;
    stMcStatusGearInMultiMaster: ST_McStatus;

    //Variables for holding limits during homing
    bWaitForStopAfterLimitHit: BOOL := FALSE;
    fbRemovePowerTimer: TOF;

    //Dedicated NC parameter read FBs
    fbReadAxisVeloManSlow: MC_ReadParameter;
    fbReadAxisVeloManFast: MC_ReadParameter;
    fbReadHomingVelToCam: MC_ReadParameter;
    fbReadHomingVelFromCam: MC_ReadParameter;
    fbReadAxisVeloMax: MC_ReadParameter;
    fbReadAxisMaxAcc: MC_ReadParameter;
    fbReadAxisMaxDec: MC_ReadParameter;
    fbReadAxisAcc: MC_ReadParameter;
    fbReadAxisDec: MC_ReadParameter;
    fbReadEnMinSoftPosLimit: MC_ReadParameter;
    fbReadEnMaxSoftPosLimit: MC_ReadParameter;
    fbReadMinSoftPosLimit: MC_ReadParameter;
    fbReadMaxSoftPosLimit: MC_ReadParameter;
    fbReadEnPositionLagMonitoring: MC_ReadParameter;
    fbReadAxisMaxPosLagValue: MC_ReadParameter;
    fbReadEnTargetPositionMonitoring: MC_ReadParameter;
    fbReadTargetPositionWindow: MC_ReadParameter;

    //Edge detection triggers for statuses
    fbDoneRTrig: R_TRIG;
    fbErrorRTrig: R_TRIG;
    fbCommandAbortedRTrig: R_TRIG;
    fbInVelocityRTrig: R_TRIG;
    fbInVelocityFTrig: F_TRIG;
    fbExecuteRTrig: R_TRIG;
    fbStopFinishedRiseEdge: R_TRIG;
    fbHaltFinishedRiseEdge: R_TRIG;
    fbResetFinishedRiseEdge: R_TRIG;
    fbAbsMovDyn1RiseEdge: R_TRIG;
    fbAbsMovDyn2RiseEdge: R_TRIG;
    fbModMovDyn1RiseEdge: R_TRIG;
    fbModMovDyn2RiseEdge: R_TRIG;

END_VAR
VAR CONSTANT
    nRATIO_DENOMINATOR_DEFAULT: UINT := 1;
    nNO_GEARING: UINT := 0;
    nMCSTATUS_ARRAY_SIZE: UINT := 13;
    nMULTI_MASTER_MAX_AXES: UINT := 4;
END_VAR

METHOD EndOfCycle : BOOL

_stAxis.stControl.bExecute := FALSE;
END_METHOD

METHOD FB_init : BOOL
VAR_INPUT
    bInitRetains: BOOL; // if TRUE, the retain variables are initialized (warm start / cold start)
    bInCopyCode: BOOL; // if TRUE, the instance afterwards gets moved into the copy code (online change)
END_VAR

//Copy address locations for statuses to an array to allow for easier checking of statuses
astMcStatus[1] := ADR(stMcStatusPower);
astMcStatus[2] := ADR(stMcStatusStop);
astMcStatus[3] := ADR(stMcStatusHalt);
astMcStatus[4] := ADR(stMcStatusReset);
astMcStatus[5] := ADR(stMcStatusMoveAbsolute);
astMcStatus[6] := ADR(stMcStatusMoveRelative);
astMcStatus[7] := ADR(stMcStatusMoveVelocity);
astMcStatus[8] := ADR(stMcStatusMoveModulo);
astMcStatus[9] := ADR(stMcStatusHome);
astMcStatus[10] := ADR(stMcStatusGearInMultiMaster);
astMcStatus[11] := ADR(stMcStatusGearOut);
astMcStatus[12] := ADR(stMcStatusReadParameter);
astMcStatus[13] := ADR(stMcStatusWriteParameter);
END_METHOD

METHOD mControl_GearInMultiMaster : ST_McStatus

fbGearInMultiMaster.Options.AdvancedSlaveDynamics := TRUE;
fbGearInMultiMaster.Options.SyncMode := E_GearInMultiMasterSyncMode.POSSYNC2;
IF _stAxis.stControl.eCommand = E_MotionFunctions.eGearInMultiMaster THEN
    fbGearInMultiMaster.Enable := _stAxis.stControl.bExecute;
END_IF

IF _stAxis.stControl.eCommand = E_MotionFunctions.eGearInMultiMaster AND _stAxis.stControl.bExecute AND NOT _stAxis.Axis.Status.Coupled THEN
    //Latch master references
    FOR nMultiMastersAxesIndex := 1 TO nMULTI_MASTER_MAX_AXES DO
        IF _stAxis.stConfig.astMultiMasterAxis[nMultiMastersAxesIndex].nIndex > 0 AND _stAxis.stConfig.astMultiMasterAxis[nMultiMastersAxesIndex].nIndex <= GVL_APP.nAXIS_NUM THEN
            _stAxis.stConfig.astMultiMasterAxisLatched[nMultiMastersAxesIndex].nIndex := _stAxis.stConfig.astMultiMasterAxis[nMultiMastersAxesIndex].nIndex;
        END_IF
    END_FOR
    //Latch gear ratios
    FOR nMultiMastersAxesIndex := 1 TO nMULTI_MASTER_MAX_AXES DO
        _stAxis.stConfig.astMultiMasterAxisLatched[nMultiMastersAxesIndex].fRatio := _stAxis.stConfig.astMultiMasterAxis[nMultiMastersAxesIndex].fRatio;
    END_FOR
    //Transfer gear ratios to FB
    fbGearInMultiMaster.GearRatio1 := _stAxis.stConfig.astMultiMasterAxisLatched[1].fRatio;
    fbGearInMultiMaster.GearRatio2 := _stAxis.stConfig.astMultiMasterAxisLatched[2].fRatio;
    fbGearInMultiMaster.GearRatio3 := _stAxis.stConfig.astMultiMasterAxisLatched[3].fRatio;
    fbGearInMultiMaster.GearRatio4 := _stAxis.stConfig.astMultiMasterAxisLatched[4].fRatio;
    fbGearInMultiMaster.Enable := TRUE;
END_IF

fbGearInMultiMaster(Slave := _stAxis.Axis,
    Master1 := GVL.astAxes[_stAxis.stConfig.astMultiMasterAxisLatched[1].nIndex].Axis,
    Master2 := GVL.astAxes[_stAxis.stConfig.astMultiMasterAxisLatched[2].nIndex].Axis,
    Master3 := GVL.astAxes[_stAxis.stConfig.astMultiMasterAxisLatched[3].nIndex].Axis,
    Master4 := GVL.astAxes[_stAxis.stConfig.astMultiMasterAxisLatched[4].nIndex].Axis);
fbGearInMultiMaster.Enable:= FALSE;

IF fbGearInMultiMaster.InGear THEN
    mStatus_MultiGearing();
END_IF

IF fbGearInMultiMaster.Error THEN
    fbGearInMultiMaster.Enable := FALSE;
END_IF

mControl_GearInMultiMaster.Active := fbGearInMultiMaster.Active;
mControl_GearInMultiMaster.Done := fbGearInMultiMaster.InGear;
mControl_GearInMultiMaster.Busy := fbGearInMultiMaster.Busy;
mControl_GearInMultiMaster.Error := fbGearInMultiMaster.Error;
mControl_GearInMultiMaster.ErrorID := fbGearInMultiMaster.ErrorID;
mControl_GearInMultiMaster.CommandAborted := fbGearInMultiMaster.CommandAborted;

IF fbGearInMultiMaster.Error THEN
    _stAxis.stError.nGearInMultiMasterErrorID := fbGearInMultiMaster.ErrorID; //Set the error
END_IF
END_METHOD

METHOD mControl_GearOut : ST_McStatus

IF _stAxis.stControl.eCommand = E_MotionFunctions.eGearOut THEN
    fbGearOut.Execute := _stAxis.stControl.bExecute;
END_IF

fbGearOut(Slave := _stAxis.Axis);
fbGearOut.Execute := FALSE;

//Clear ratios from single and multi master gearing
IF fbGearOut.Done THEN
    //Clear slave ratio from master axis slave array
    mStatus_MultiGearing();
    FOR nSlaveAxesIndex := 1 TO GVL_APP.nAXIS_NUM DO
        GVL.astAxes[nSlaveAxesIndex].stConfig.afMultiSlaveAxisRatio[GVL.iAxis] := nNO_GEARING;
    END_FOR
END_IF

mControl_GearOut.Done := fbGearOut.Done;
mControl_GearOut.Busy := fbGearOut.Busy;
mControl_GearOut.Error := fbGearOut.Error;
mControl_GearOut.ErrorID := fbGearOut.ErrorID;

IF fbGearOut.Error THEN
    _stAxis.stError.nGearOutErrorID := fbGearOut.ErrorID; //Set the error
END_IF
END_METHOD

METHOD mControl_Home : ST_McStatus
IF _stAxis.stConfig.eHomeSeq = E_HomingRoutines.eNoHoming THEN
    _stAxis.stStatus.bHomed := TRUE;
END_IF

IF _stAxis.stControl.eCommand = E_MotionFunctions.eHome THEN
    fbHome.bExecute := _stAxis.stControl.bExecute;
END_IF


fbHome.eHomeSeq := _stAxis.stConfig.eHomeSeq;
fbHome.fHomePosition := _stAxis.stConfig.fHomePosition;
fbHome.fHomeFinishDistance := _stAxis.stConfig.fHomeFinishDistance;
fbHome(
    Axis := _stAxis.Axis,
    bLimitBwd := _stAxis.stInputs.bLimitBwd,
    bLimitFwd := _stAxis.stInputs.bLimitFwd,
    bHomeSensor := _stAxis.stInputs.bHomeSensor,
    stConfig := _stAxis.stConfig);
fbHome.bExecute := FALSE;

mControl_Home.Busy := fbHome.bBusy;
mControl_Home.CommandAborted := fbHome.bCommandAborted;
mControl_Home.Done := fbHome.bDone;
mControl_Home.Error := fbHome.bError;
mControl_Home.ErrorID := fbHome.nErrorId;

IF fbHome.bError THEN
    _stAxis.stError.nHomeErrorID := fbHome.nErrorID; //Set the error
END_IF
END_METHOD

METHOD mControl_LimitHitTimer : BOOL

//Timer for keeping power on after limit switch hit, needed for homing routines - if power is lost routines are aborted
fbRemovePowerTimer(IN := _stAxis.stInputs.bLimitFwd AND _stAxis.stInputs.bLimitBwd, PT := T#100MS);

IF stMcStatusHome.Busy AND (fbRemovePowerTimer.Q OR _stAxis.Axis.NcToPlc.AxisState = 5) THEN //5=PHASE_ACCNEG
    bWaitForStopAfterLimitHit := TRUE;
ELSE
    bWaitForStopAfterLimitHit := FALSE;
END_IF
END_METHOD

METHOD mControl_LimitLinking : BOOL

_stAxis.stStatus.bFwEnabled := _stAxis.stInputs.bLimitFwd; //Moved to linking code. Should not say enabled if not enabled
_stAxis.stStatus.bBwEnabled := _stAxis.stInputs.bLimitBwd;
_stAxis.stStatus.bInterlockedFwd := _stAxis.stControl.bInterlockFwd;
_stAxis.stStatus.bInterlockedBwd := _stAxis.stControl.bInterlockBwd;

//Multimaster limit linking
FOR nAxisIndex := 1 TO GVL_APP.nAXIS_NUM DO
    IF (_stAxis.stConfig.afMultiSlaveAxisRatio[nAxisIndex] <> 0) THEN
        _stAxis.stStatus.bFwEnabled := _stAxis.stStatus.bFwEnabled AND SEL(_stAxis.stConfig.afMultiSlaveAxisRatio[nAxisIndex] > 0, GVL.astAxes[nAxisIndex].stStatus.bBwEnabled, GVL.astAxes[nAxisIndex].stStatus.bFwEnabled);
        _stAxis.stStatus.bBwEnabled := _stAxis.stStatus.bBwEnabled AND SEL(_stAxis.stConfig.afMultiSlaveAxisRatio[nAxisIndex] > 0, GVL.astAxes[nAxisIndex].stStatus.bFwEnabled, GVL.astAxes[nAxisIndex].stStatus.bBwEnabled);
    END_IF
END_FOR
END_METHOD

METHOD mControl_Power : ST_McStatus
VAR
END_VAR
IF mControl_TemperatureDisable(_stAxis.stConfig.bEnableTemperatureDisable) THEN
    _stAxis.stControl.bEnable:= FALSE;
END_IF

fbPower.Enable := _stAxis.stControl.bEnable;

fbPower.Enable_Negative := (_stAxis.stStatus.bBwEnabled OR bWaitForStopAfterLimitHit) AND NOT _stAxis.stStatus.bInterlockedBwd;
fbPower.Enable_Positive := (_stAxis.stStatus.bFwEnabled OR bWaitForStopAfterLimitHit) AND NOT _stAxis.stStatus.bInterlockedFwd;
fbPower.Override := _stAxis.stConfig.fOverride;

fbPower(Axis := _stAxis.Axis);

mControl_Power.Error := fbPower.Error;

IF fbPower.Error THEN
    _stAxis.stError.nPowerErrorID := fbPower.ErrorID; //Set the error
END_IF
END_METHOD

METHOD mControl_Reset : ST_McStatus
VAR
    i: UINT;
END_VAR
fbReset.Execute := _stAxis.stControl.bReset;

fbReset(Axis := _stAxis.Axis);
IF fbReset.Done THEN
    _stAxis.stStatus.bError := FALSE;
    FOR i := 1 TO nMCSTATUS_ARRAY_SIZE DO
        //Reset ST_Status error ID
        _stAxis.stStatus.nErrorID := 0;
        //Reset St_AxisError error IDs
        _stAxis.stError.nPowerErrorID := 0;
        _stAxis.stError.nMoveAbsoluteErrorID := 0;
        _stAxis.stError.nMoveRelativeErrorID := 0;
        _stAxis.stError.nMoveVelocityErrorID := 0;
        _stAxis.stError.nMoveModuloErrorID := 0;
        _stAxis.stError.nHomeErrorID := 0;
        _stAxis.stError.nHaltErrorID := 0;
        _stAxis.stError.nResetErrorID := 0;
        _stAxis.stError.nStopErrorID := 0;
        _stAxis.stError.nGearInMultiMasterErrorID := 0;
        _stAxis.stError.nGearOutErrorID := 0;
        _stAxis.stError.nWriteParameterErrorId := 0;
        _stAxis.stError.nReadParameterErrorId := 0;
        _stAxis.stError.nNCErrorID := 0;
    END_FOR
END_IF

mControl_Reset.Busy := fbReset.Busy;
mControl_Reset.Done := fbReset.Done;
mControl_Reset.Error := fbReset.Error;
mControl_Reset.ErrorID := fbReset.ErrorID;

IF fbReset.Error THEN
    _stAxis.stError.nResetErrorID := fbReset.ErrorID; //Set the error
END_IF

fbResetFinishedRiseEdge(CLK:=fbReset.Done OR fbReset.Error);
IF fbResetFinishedRiseEdge.Q OR fbReset.Done THEN
    _stAxis.stControl.bReset := FALSE;
END_IF
END_METHOD

METHOD mControl_TemperatureDisable: BOOL
VAR_INPUT
    bEnableTemperatureDisable: BOOL;
END_VAR
VAR
    nAxisId: UINT;
    fTemperatureScaledValue: LREAL;
    fTemperatureValue: LREAL;
    sErrorMessage: STRING(255);
    sErrorMessageAxis: STRING;
END_VAR
VAR_INST
    fbErrorTrig: R_TRIG;
    fbErrorTON: TON;
    fMAX_TEMP_LIMIT: LREAL := 850.0;
    fMIN_TEMP_LIMIT: LREAL := -200.0;
    bError: BOOL := FALSE;
END_VAR
nAxisId := DWORD_TO_UINT(_stAxis.Axis.NcToPlc.AxisId);
sErrorMessageAxis := CONCAT('ERROR: Temparture sensor of axis ',UINT_TO_STRING(nAxisId));
fbErrorTrig(clk:=bError);
fTemperatureScaledValue := INT_TO_LREAL(_stAxis.stInputs.nTempPT100)/_stAxis.stConfig.fTempScalingFactor;
fTemperatureValue := SEL(_stAxis.stControl.bHWMaskActive,fTemperatureScaledValue,_stAxis.stControl.fMaskedTemperature);
fbErrorTON(in:=bError, PT:=T#30S);

IF bEnableTemperatureDisable THEN
    //Check for disconnection or wrongly connected errors
    IF fTemperatureValue >= fMAX_TEMP_LIMIT OR fTemperatureValue <= fMIN_TEMP_LIMIT THEN
        _stAxis.stStatus.fActTemperature := fTemperatureValue;
        _stAxis.stStatus.bHighTempAxisDisabled := TRUE;
        bError := TRUE;

        IF fbErrorTrig.Q THEN
            IF fTemperatureValue = fMAX_TEMP_LIMIT THEN
                sErrorMessage := CONCAT(sErrorMessageAxis,' is disconnected.');
                ADSLOGSTR( msgCtrlMask := ADSLOG_MSGTYPE_ERROR, msgFmtStr := '%s', strArg := sErrorMessage);
            ELSIF fTemperatureValue = fMIN_TEMP_LIMIT THEN
                sErrorMessage := CONCAT(sErrorMessageAxis,' is wrongly connected, check PT100 pin connections.');
                ADSLOGSTR( msgCtrlMask := ADSLOG_MSGTYPE_ERROR, msgFmtStr := '%s', strArg := sErrorMessage);
            END_IF
        END_IF

        //Reset bError to display Error message every 10 seconds if error is still there
        IF fbErrorTON.Q THEN
            bError := FALSE;
        END_IF

        mControl_TemperatureDisable := TRUE;
        RETURN;
    END_IF

    //Check scaled tempearture value agianst max. allowed temperature
    IF fTemperatureValue < _stAXis.stConfig.fMaxTemperature THEN
        bError := FALSE;
        sErrorMessage := '';
        _stAxis.stStatus.fActTemperature := fTemperatureValue;
        _stAxis.stStatus.bHighTempAxisDisabled := FALSE;
        mControl_TemperatureDisable := FALSE;
        RETURN;
    ELSIF fTemperatureValue >= _stAXis.stConfig.fMaxTemperature THEN
        bError := TRUE;
        _stAxis.stStatus.fActTemperature := fTemperatureValue;
        _stAxis.stStatus.bHighTempAxisDisabled := TRUE;
        IF fbErrorTrig.Q THEN
            sErrorMessage := CONCAT('ERROR: Axis temperature too hot. Cannot enable Axis ',UINT_TO_STRING(nAxisId));
            ADSLOGSTR( msgCtrlMask := ADSLOG_MSGTYPE_ERROR, msgFmtStr := '%s', strArg := sErrorMessage);
        END_IF

        IF fbErrorTON.Q THEN
            bError := FALSE;
        END_IF
        mControl_TemperatureDisable := TRUE;
        RETURN;
    END_IF
ELSE
    _stAxis.stStatus.fActTemperature := fTemperatureValue;
    _stAxis.stStatus.bHighTempAxisDisabled := FALSE;
    mControl_TemperatureDisable := FALSE;
    RETURN;
END_IF
END_METHOD

METHOD mMove_Halt : ST_McStatus

fbHalt.Deceleration := _stAxis.stControl.fDeceleration;
fbHalt.Execute := _stAxis.stControl.bHalt;

fbHalt(Axis := _stAxis.Axis);

mMove_Halt.Busy := fbHalt.Busy;
mMove_Halt.Done := fbHalt.Done;
mMove_Halt.Error := fbHalt.Error;
mMove_Halt.ErrorID := fbHalt.ErrorID;
mMove_Halt.Active := fbHalt.Active;
mMove_Halt.CommandAborted := fbHalt.CommandAborted;

IF fbHalt.Error THEN
    _stAxis.stError.nHaltErrorID := fbHalt.ErrorID; //Set the error
END_IF

//Execution of fbHalt ended
fbHaltFinishedRiseEdge(CLK:=fbHalt.Done OR fbHalt.Error OR fbHalt.CommandAborted);
IF fbHaltFinishedRiseEdge.Q OR fbHalt.Done OR fbHalt.CommandAborted THEN
    _stAxis.stControl.bHalt := FALSE;
END_IF
END_METHOD

METHOD mMove_MoveAbsolute : ST_McStatus
IF _stAxis.stControl.eCommand = E_MotionFunctions.eMoveAbsolute THEN
    fbMoveAbsolute.Execute := _stAxis.stControl.bExecute;
    IF fbMoveAbsolute.Execute AND fbMoveAbsolute.Busy THEN
        fbMoveAbsolute2.Execute := TRUE;
    END_IF
END_IF

// Parameters
fbMoveAbsolute.Position := _stAxis.stControl.fPosition;
fbMoveAbsolute.Velocity := ABS(_stAxis.stControl.fVelocity);
fbMoveAbsolute.Acceleration := _stAxis.stControl.fAcceleration;
fbMoveAbsolute.Deceleration := _stAxis.stControl.fDeceleration;

fbMoveAbsolute2.Position := _stAxis.stControl.fPosition;
fbMoveAbsolute2.Velocity := ABS(_stAxis.stControl.fVelocity);
fbMoveAbsolute2.Acceleration := _stAxis.stControl.fAcceleration;
fbMoveAbsolute2.Deceleration := _stAxis.stControl.fDeceleration;


// Call both move absolute FB
fbMoveAbsolute(Axis := _stAxis.Axis);
fbMoveAbsolute2(Axis := _stAxis.Axis);

//Reset Execute bits
fbMoveAbsolute.Execute := FALSE;
fbMoveAbsolute2.Execute := FALSE;


// STATUS bits
mMove_MoveAbsolute.Active := fbMoveAbsolute.Active OR fbMoveAbsolute2.Active;
mMove_MoveAbsolute.Done := fbMoveAbsolute.Done OR fbMoveAbsolute2.Done;
mMove_MoveAbsolute.Busy := fbMoveAbsolute.Busy OR fbMoveAbsolute2.Busy;
mMove_MoveAbsolute.Error := fbMoveAbsolute.Error OR fbMoveAbsolute2.Error;


// Capture the CommandAborted for first scan if the other absolute move overtakes the current
fbAbsMovDyn1RiseEdge(CLK:= fbMoveAbsolute.Busy AND fbMoveAbsolute2.CommandAborted, Q=>);
fbAbsMovDyn2RiseEdge(CLK:= fbMoveAbsolute2.Busy AND fbMoveAbsolute.CommandAborted, Q=>);
mMove_MoveAbsolute.CommandAborted := (fbMoveAbsolute.CommandAborted AND NOT fbAbsMovDyn2RiseEdge.Q)
                                    OR (fbMoveAbsolute2.CommandAborted AND NOT fbAbsMovDyn1RiseEdge.Q);

// Error IDs
IF fbMoveAbsolute.Error THEN
    _stAxis.stError.nMoveAbsoluteErrorID := fbMoveAbsolute.ErrorID; //Set the error
    mMove_MoveAbsolute.ErrorID := fbMoveAbsolute.ErrorID;
END_IF
IF fbMoveAbsolute2.Error THEN
    _stAxis.stError.nMoveAbsoluteErrorID := fbMoveAbsolute2.ErrorID; //Set the error
    mMove_MoveAbsolute.ErrorID := fbMoveAbsolute2.ErrorID;
END_IF
END_METHOD

METHOD mMove_MoveModulo : ST_McStatus
IF _stAxis.stControl.eCommand = E_MotionFunctions.eMoveModulo THEN
    fbMoveModulo.Execute := _stAxis.stControl.bExecute;
    IF fbMoveModulo.Execute AND fbMoveModulo.Busy THEN
        fbMoveModulo2.Execute := TRUE;
    END_IF
END_IF

// Parameters
fbMoveModulo.Position := _stAxis.stControl.fPosition;
fbMoveModulo.Velocity := ABS(_stAxis.stControl.fVelocity);
fbMoveModulo.Acceleration := _stAxis.stControl.fAcceleration;
fbMoveModulo.Deceleration := _stAxis.stControl.fDeceleration;

fbMoveModulo2.Position := _stAxis.stControl.fPosition;
fbMoveModulo2.Velocity := ABS(_stAxis.stControl.fVelocity);
fbMoveModulo2.Acceleration := _stAxis.stControl.fAcceleration;
fbMoveModulo2.Deceleration := _stAxis.stControl.fDeceleration;

// Call both move absolute FB
fbMoveModulo(Axis := _stAxis.Axis);
fbMoveModulo.Execute := FALSE;
fbMoveModulo2(Axis := _stAxis.Axis);
fbMoveModulo2.Execute := FALSE;

// Status bits
mMove_MoveModulo.Active := fbMoveModulo.Active OR fbMoveModulo2.Active;
mMove_MoveModulo.Done := fbMoveModulo.Done OR fbMoveModulo2.Done;
mMove_MoveModulo.Busy := fbMoveModulo.Busy OR fbMoveModulo2.Busy;
mMove_MoveModulo.Error := fbMoveModulo.Error OR fbMoveModulo2.Error;

// Capture the CommandAborted for first scan if the other absolute move overtakes the current
fbModMovDyn1RiseEdge(CLK:= fbMoveModulo.Busy AND fbMoveModulo2.CommandAborted, Q=>);
fbModMovDyn2RiseEdge(CLK:= fbMoveModulo2.Busy AND fbMoveModulo.CommandAborted, Q=>);
mMove_MoveModulo.CommandAborted := (fbMoveModulo.CommandAborted AND NOT fbModMovDyn2RiseEdge.Q)
                                    OR (fbMoveModulo2.CommandAborted AND NOT fbModMovDyn1RiseEdge.Q);

// Error IDs
IF fbMoveModulo.Error THEN
    _stAxis.stError.nMoveModuloErrorID := fbMoveModulo.ErrorID; //Set the error
    mMove_MoveModulo.ErrorID := fbMoveModulo.ErrorID;
END_IF

IF fbMoveModulo2.Error THEN
    _stAxis.stError.nMoveModuloErrorID := fbMoveModulo2.ErrorID; //Set the error
    mMove_MoveModulo.ErrorID := fbMoveModulo2.ErrorID;
END_IF
END_METHOD

METHOD mMove_MoveRelative : ST_McStatus

IF _stAxis.stControl.eCommand = E_MotionFunctions.eMoveRelative THEN
    fbMoveRelative.Execute := _stAxis.stControl.bExecute;
END_IF

fbMoveRelative.Distance := _stAxis.stControl.fPosition;
fbMoveRelative.Velocity := ABS(_stAxis.stControl.fVelocity);
fbMoveRelative.Acceleration := _stAxis.stControl.fAcceleration;
fbMoveRelative.Deceleration := _stAxis.stControl.fDeceleration;

fbMoveRelative(Axis := _stAxis.Axis);
fbMoveRelative.Execute := FALSE;

mMove_MoveRelative.Active := fbMoveRelative.Active;
mMove_MoveRelative.Done := fbMoveRelative.Done;
mMove_MoveRelative.Busy := fbMoveRelative.Busy;
mMove_MoveRelative.Error := fbMoveRelative.Error;
mMove_MoveRelative.ErrorID := fbMoveRelative.ErrorID;
mMove_MoveRelative.CommandAborted := fbMoveRelative.CommandAborted;

IF fbMoveRelative.Error THEN
    _stAxis.stError.nMoveRelativeErrorID := fbMoveRelative.ErrorID; //Set the error
END_IF
END_METHOD

METHOD mMove_MoveVelocity : ST_McStatus

IF _stAxis.stControl.eCommand = E_MotionFunctions.eMoveVelocity THEN
    fbMoveVelocity.Execute := _stAxis.stControl.bExecute;
END_IF

fbMoveVelocity.Direction := SEL(_stAxis.stControl.fVelocity < 0, MC_Positive_Direction, MC_Negative_Direction);
fbMoveVelocity.Velocity := ABS(_stAxis.stControl.fVelocity);
fbMoveVelocity.Acceleration := _stAxis.stControl.fAcceleration;
fbMoveVelocity.Deceleration := _stAxis.stControl.fDeceleration;

fbMoveVelocity(Axis := _stAxis.Axis);
fbMoveVelocity.Execute:= FALSE;

mMove_MoveVelocity.Active := fbMoveVelocity.Active;
mMove_MoveVelocity.InVelocity := fbMoveVelocity.InVelocity;
mMove_MoveVelocity.Busy := fbMoveVelocity.Busy;
mMove_MoveVelocity.Error := fbMoveVelocity.Error;
mMove_MoveVelocity.ErrorID := fbMoveVelocity.ErrorID;
mMove_MoveVelocity.CommandAborted := fbMoveVelocity.CommandAborted;

IF fbMoveVelocity.Error THEN
    _stAxis.stError.nMoveVelocityErrorID := fbMoveVelocity.ErrorID; //Set the error
END_IF
END_METHOD

METHOD mMove_Stop : ST_McStatus

fbStop.Deceleration := _stAxis.stControl.fDeceleration;
fbStop.Execute := _stAxis.stControl.bStop;

fbStop(Axis := _stAxis.Axis);

mMove_Stop.Busy := fbStop.Busy;
mMove_Stop.Done := fbStop.Done;
mMove_Stop.Error := fbStop.Error;
mMove_Stop.ErrorID := fbStop.ErrorID;
mMove_Stop.Active := fbStop.Active;
mMove_Stop.CommandAborted := fbStop.CommandAborted;

IF fbStop.Error THEN
    _stAxis.stError.nStopErrorID := fbStop.ErrorID; //Set the error
END_IF

//Execution of fbStop ended
fbStopFinishedRiseEdge(CLK:=fbStop.Done OR fbStop.Error OR fbStop.CommandAborted);
IF fbStopFinishedRiseEdge.Q THEN
    _stAxis.stControl.bStop := FALSE;
END_IF
END_METHOD

METHOD mParameters_Init : BOOL

IF _stAxis.stConfig.bReadMcParametersValid AND NOT _stAxis.stStatus.bAxisInitialized THEN
    _stAxis.stControl.fAcceleration := _stAxis.stConfig.fDefaultAcc;
    _stAxis.stControl.fDeceleration := _stAxis.stConfig.fDefaultDec;
    _stAxis.stControl.fVelocity := _stAxis.stConfig.fVelocityDefaultFast;
    _stAxis.stControl.fJogVelocity := _stAxis.stConfig.fVelocityDefaultSlow;

    _stAxis.stStatus.bAxisInitialized := TRUE;
END_IF
END_METHOD

METHOD mParameters_ReadNc : BOOL

(*This act reads the MC parameters using an MC_ReadParameter FB FOR each variable
Intended TO be executed once every PLC cycle
Another FB is used TO trasnfer default axis parameters TO the stAxisStruct so
bReadValid is used TO halt that trasnfer UNTIL the parameters have been
read successfully. It may take a couple OF cycles once the PLC starts up.*)

//Slow jogging Velocity
fbReadAxisVeloManSlow(Axis := _stAxis.Axis,
                        Enable := TRUE,
                        ReadMode := READMODE_CYCLIC,
                        ParameterNumber := E_AxisParameters.AxisManualVelocitySlow,
                        Value => _stAxis.stConfig.fVelocityDefaultSlow);
//Fast jogging velocity
fbReadAxisVeloManFast(Axis := _stAxis.Axis,
                        Enable := TRUE,
                        ReadMode := READMODE_CYCLIC,
                        ParameterNumber := E_AxisParameters.AxisManualVelocityFast,
                        Value => _stAxis.stConfig.fVelocityDefaultFast);
//Homing velocity to Cam
fbReadHomingVelToCam(Axis := _stAxis.Axis,
                        Enable := TRUE,
                        ReadMode := READMODE_CYCLIC,
                        ParameterNumber := E_AxisParameters.AxisVelocityToCam,
                        Value => _stAxis.stConfig.fHomingVelToCam);
//Homing velocity from Cam
fbReadHomingVelFromCam(Axis := _stAxis.Axis,
                        Enable := TRUE,
                        ReadMode := READMODE_CYCLIC,
                        ParameterNumber := E_AxisParameters.AxisVelocityFromCam,
                        Value => _stAxis.stConfig.fHomingVelFromCam);
//Max velocity
fbReadAxisVeloMax(Axis := _stAxis.Axis,
                        Enable := TRUE,
                        ReadMode := READMODE_CYCLIC,
                        ParameterNumber := E_AxisParameters.AxisMaxVelocity,
                        Value => _stAxis.stConfig.fVeloMax);
//Max acceleration
fbReadAxisMaxAcc(Axis := _stAxis.Axis,
                        Enable := TRUE,
                        ReadMode := READMODE_CYCLIC,
                        ParameterNumber := E_AxisParameters.AxisMaximumAcceleration,
                        Value => _stAxis.stConfig.fMaxAcc);
//Max deceleration
fbReadAxisMaxDec(Axis := _stAxis.Axis,
                        Enable := TRUE,
                        ReadMode := READMODE_CYCLIC,
                        ParameterNumber := E_AxisParameters.AxisMaximumDeceleration,
                        Value => _stAxis.stConfig.fMaxDec);
//Default acceleration
fbReadAxisAcc(Axis := _stAxis.Axis,
                        Enable := TRUE,
                        ReadMode := READMODE_CYCLIC,
                        ParameterNumber := E_AxisParameters.AxisDefaultAcceleration,
                        Value => _stAxis.stConfig.fDefaultAcc);
//Default deceleration
fbReadAxisDec(Axis := _stAxis.Axis,
                        Enable := TRUE,
                        ReadMode := READMODE_CYCLIC,
                        ParameterNumber := E_AxisParameters.AxisDefaultDeceleration,
                        Value => _stAxis.stConfig.fDefaultDec);

//Soft limits enabled
fbReadEnMinSoftPosLimit(Axis := _stAxis.Axis,
                        Enable := TRUE,
                        ReadMode := READMODE_CYCLIC,
                        ParameterNumber := E_AxisParameters.EnableLimitBackward);
_stAxis.stConfig.bEnMinSoftPosLimit := LREAL_TO_BOOL(fbReadEnMinSoftPosLimit.Value);

fbReadEnMaxSoftPosLimit(Axis := _stAxis.Axis,
                        Enable := TRUE,
                        ReadMode := READMODE_CYCLIC,
                        ParameterNumber := E_AxisParameters.EnableLimitForward);
_stAxis.stConfig.bEnMaxSoftPosLimit := LREAL_TO_BOOL(fbReadEnMaxSoftPosLimit.Value);

//Soft limit values
fbReadMinSoftPosLimit(Axis := _stAxis.Axis,
                        Enable := TRUE,
                        ReadMode := READMODE_CYCLIC,
                        ParameterNumber := E_AxisParameters.SWLimitBackward,
                        Value => _stAxis.stConfig.fMinSoftPosLimit);
fbReadMaxSoftPosLimit(Axis := _stAxis.Axis,
                        Enable := TRUE,
                        ReadMode := READMODE_CYCLIC,
                        ParameterNumber := E_AxisParameters.SWLimitForward,
                        Value => _stAxis.stConfig.fMaxSoftPosLimit);

//Position Lag Monitoring
fbReadEnPositionLagMonitoring(Axis := _stAxis.Axis,
                        Enable := TRUE,
                        ReadMode := READMODE_CYCLIC,
                        ParameterNumber := E_AxisParameters.EnablePositionLagMonitoring);
_stAxis.stConfig.bEnPositionLagMonitoring := LREAL_TO_BOOL(fbReadEnPositionLagMonitoring.Value);

fbReadAxisMaxPosLagValue(Axis := _stAxis.Axis,
                        Enable := TRUE,
                        ReadMode := READMODE_CYCLIC,
                        ParameterNumber := E_AxisParameters.MaxPositionLag,
                        Value => _stAxis.stConfig.fMaxPosLagValue);

// Target Position Monitoring
fbReadEnTargetPositionMonitoring(Axis := _stAxis.Axis,
                        Enable := TRUE,
                        ReadMode := READMODE_CYCLIC,
                        ParameterNumber := E_AxisParameters.SWLimitBackward);
_stAxis.stConfig.bEnTargetPositionMonitoring := LREAL_TO_BOOL(fbReadEnTargetPositionMonitoring.Value);

fbReadTargetPositionWindow(Axis := _stAxis.Axis,
                        Enable := TRUE,
                        ReadMode := READMODE_CYCLIC,
                        ParameterNumber := E_AxisParameters.AxisTargetPositionWindow,
                        Value => _stAxis.stConfig.fTargetPositionWindow);

//All variables are valid
_stAxis.stConfig.bReadMcParametersValid := FALSE;
_stAxis.stConfig.bReadMcParametersValid := fbReadAxisVeloManSlow.Valid AND
    fbReadAxisVeloManFast.Valid AND
    fbReadHomingVelToCam.Valid AND
    fbReadHomingVelFromCam.Valid AND
    fbReadAxisVeloMax.Valid AND
    fbReadAxisAcc.Valid AND
    fbReadAxisDec.Valid AND
    fbReadEnMinSoftPosLimit.Valid AND
    fbReadEnMaxSoftPosLimit.Valid AND
    fbReadMinSoftPosLimit.Valid AND
    fbReadMaxSoftPosLimit.Valid AND
    fbReadEnPositionLagMonitoring.Valid AND
    fbReadAxisMaxPosLagValue.Valid AND
    fbReadEnTargetPositionMonitoring.Valid AND
    fbReadTargetPositionWindow.Valid;

//One of the variables has a read error
_stAxis.stConfig.bReadMcParametersError := fbReadAxisVeloManSlow.Error OR
    fbReadAxisVeloManFast.Error OR
    fbReadHomingVelToCam.Error OR
    fbReadHomingVelFromCam.Error OR
    fbReadAxisVeloMax.Error OR
    fbReadAxisAcc.Error OR
    fbReadAxisDec.Error OR
    fbReadEnMinSoftPosLimit.Error OR
    fbReadEnMaxSoftPosLimit.Error OR
    fbReadMinSoftPosLimit.Error OR
    fbReadMaxSoftPosLimit.Error OR
    fbReadEnPositionLagMonitoring.Error OR
    fbReadAxisMaxPosLagValue.Error OR
    fbReadEnTargetPositionMonitoring.Error OR
    fbReadTargetPositionWindow.Error;
END_METHOD

METHOD mParameters_ReadParameter : ST_McStatus

IF _stAxis.stControl.eCommand = E_MotionFunctions.eReadParameter THEN
    fbReadParameter.Enable := _stAxis.stControl.bExecute;
END_IF

fbReadParameter.ReadMode := E_READMODE.READMODE_ONCE;
fbReadParameter.ParameterNumber := _stAxis.stConfig.eAxisParameters;

fbReadParameter(Axis := _stAxis.Axis);
fbReadParameter.Enable := FALSE;

_stAxis.stconfig.fReadAxisParameter := fbReadParameter.Value;
mParameters_ReadParameter.Busy := fbReadParameter.Busy;
mParameters_ReadParameter.Done := fbReadParameter.Valid;
mParameters_ReadParameter.Error := fbReadParameter.Error;
mParameters_ReadParameter.ErrorID := fbReadParameter.ErrorID;

IF fbReadParameter.Error THEN
    _stAxis.stError.nReadParameterErrorId := fbReadParameter.ErrorID;
END_IF
END_METHOD

METHOD mParameters_WriteParameter : ST_McStatus

IF _stAxis.stControl.eCommand = E_MotionFunctions.eWriteParameter THEN
    fbWriteParameter.Execute := _stAxis.stControl.bExecute;
END_IF

fbWriteParameter.ParameterNumber := _stAxis.stConfig.eAxisParameters;
fbWriteParameter.Value := _stAxis.stConfig.fWriteAxisParameter;

fbWriteParameter(Axis := _stAxis.Axis);
fbWriteParameter.Execute := FALSE;

mParameters_WriteParameter.Busy := fbWriteParameter.Busy;
mParameters_WriteParameter.Done := fbWriteParameter.Done;
mParameters_WriteParameter.Error := fbWriteParameter.Error;
mParameters_WriteParameter.ErrorID := fbWriteParameter.ErrorID;

IF fbWriteParameter.Error THEN
    _stAxis.stError.nWriteParameterErrorId := fbWriteParameter.ErrorID;
END_IF
END_METHOD

METHOD mStatus_AxisStatus : BOOL

_stAxis.Axis.ReadStatus();
IF _stAxis.Axis.Status.OpMode.Modulo THEN
    _stAxis.stStatus.fActPosition := _stAxis.Axis.NcToPlc.ModuloActPos;
ELSE
    _stAxis.stStatus.fActPosition := _stAxis.Axis.NcToPlc.ActPos;
END_IF

_stAxis.stStatus.bGeared := _stAxis.Axis.Status.Coupled;
_stAxis.stStatus.bHomed := _stAxis.Axis.Status.Homed;
_stAxis.stStatus.bMoving := _stAxis.Axis.Status.Moving;
_stAxis.stStatus.fActVelocity := _stAxis.Axis.NcToPlc.ActVelo;
_stAxis.stStatus.bMovingForward := _stAxis.Axis.Status.PositiveDirection;
_stAxis.stStatus.bMovingBackward := _stAxis.Axis.Status.NegativeDirection;
_stAxis.stStatus.bInTargetPosition := _stAxis.Axis.Status.InTargetPosition;
_stAxis.stStatus.bEnabled := NOT(_stAxis.Axis.Status.Disabled);
_stAxis.stError.nNCErrorID := _stAxis.Axis.Status.ErrorID;
END_METHOD

METHOD mStatus_Busy : BOOL
VAR
    i: UINT;
    tmpBusy: BOOL;
END_VAR

FOR i := 5 TO nMCSTATUS_ARRAY_SIZE DO
    tmpBusy := astMcStatus[i]^.Busy OR tmpBusy;
END_FOR
mStatus_Busy := tmpBusy;
END_METHOD

METHOD mStatus_CommandAborted : BOOL
VAR
    i: UINT;
    tmpCmdAborted: BOOL;
END_VAR

FOR i := 5 TO nMCSTATUS_ARRAY_SIZE DO
    tmpCmdAborted := astMcStatus[i]^.CommandAborted OR tmpCmdAborted;
END_FOR

fbCommandAbortedRTrig(CLK := tmpCmdAborted);
IF fbCommandAbortedRTrig.Q THEN
    _stAxis.stStatus.bCommandAborted := TRUE;
END_IF
END_METHOD

METHOD mStatus_Done : BOOL
VAR
    i: UINT;
    tmpDone: BOOL;
END_VAR

FOR i := 5 TO nMCSTATUS_ARRAY_SIZE DO
    tmpDone := astMcStatus[i]^.Done OR tmpDone;
END_FOR
//fbDoneRTrig(CLK:= mStatus_Done());
fbDoneRTrig(CLK := tmpDone);
IF fbDoneRTrig.Q THEN
    _stAxis.stStatus.bDone := TRUE;
END_IF
END_METHOD

METHOD mStatus_Error : BOOL
VAR
    i: UINT;
    tmpError: BOOL;
END_VAR
FOR i := 1 TO nMCSTATUS_ARRAY_SIZE DO
    tmpError := astMcStatus[i]^.Error OR tmpError;
END_FOR

fbErrorRTrig(CLK := tmpError);

IF _stAxis.Axis.Status.ErrorStop THEN
    _stAxis.stStatus.bError := _stAxis.Axis.Status.ErrorStop;
    _stAxis.stStatus.nErrorID := _stAxis.Axis.Status.ErrorID;//NC Error ID
ELSIF _stAxis.Axis.Status.Error THEN
    _stAxis.stStatus.nErrorID := _stAxis.stError.nNCErrorID;
ELSIF fbErrorRTrig.Q THEN
        //For each mcStatus
        FOR i := 1 TO nMCSTATUS_ARRAY_SIZE DO
            //If there's an error present propagate
            IF astMcStatus[i]^.ErrorID <> 0 THEN
                _stAxis.stStatus.nErrorID := astMcStatus[i]^.ErrorID;
            END_IF
        END_FOR
END_IF
END_METHOD

METHOD mStatus_InVelocity : BOOL
VAR
    i: UINT;
    tmpInVelocity: BOOL;
END_VAR
FOR i := 1 TO nMCSTATUS_ARRAY_SIZE DO
    tmpInVelocity := astMcStatus[i]^.InVelocity OR tmpInVelocity;
END_FOR
//fbInVelocityRTrig(CLK:= mStatus_InVelocity());
fbInVelocityRTrig(CLK := tmpInVelocity);
IF fbInVelocityRTrig.Q THEN
    _stAxis.stStatus.bInVelocity := TRUE;
END_IF

fbInVelocityFTrig(CLK := _stAxis.Axis.Status.ContinuousMotion);
IF fbInVelocityFTrig.Q THEN
    _stAxis.stStatus.bInVelocity := FALSE;
END_IF
END_METHOD

METHOD mStatus_MultiGearing : BOOL

IF _stAxis.Axis.Status.Coupled AND _stAxis.Axis.PlcToNc.GearRatio1 <> 0 AND _stAxis.stConfig.astMultiMasterAxisLatched[1].nIndex <> 0 THEN
    GVL.astAxes[_stAxis.stConfig.astMultiMasterAxisLatched[1].nIndex].stConfig.afMultiSlaveAxisRatio[GVL.iAxis] := _stAxis.Axis.PlcToNc.GearRatio1;
    _stAxis.stStatus.bCoupledGear1 := TRUE;
ELSE
    _stAxis.stStatus.bCoupledGear1 := FALSE;
END_IF

IF _stAxis.Axis.Status.Coupled AND _stAxis.Axis.PlcToNc.GearRatio2 <> 0 AND _stAxis.stConfig.astMultiMasterAxisLatched[2].nIndex <> 0 THEN
    GVL.astAxes[_stAxis.stConfig.astMultiMasterAxisLatched[2].nIndex].stConfig.afMultiSlaveAxisRatio[GVL.iAxis] := _stAxis.Axis.PlcToNc.GearRatio2;
    _stAxis.stStatus.bCoupledGear2 := TRUE;
ELSE
    _stAxis.stStatus.bCoupledGear2 := FALSE;
END_IF

IF _stAxis.Axis.Status.Coupled AND _stAxis.Axis.PlcToNc.GearRatio3 <> 0 AND _stAxis.stConfig.astMultiMasterAxisLatched[3].nIndex <> 0 THEN
    GVL.astAxes[_stAxis.stConfig.astMultiMasterAxisLatched[3].nIndex].stConfig.afMultiSlaveAxisRatio[GVL.iAxis] := _stAxis.Axis.PlcToNc.GearRatio3;
    _stAxis.stStatus.bCoupledGear3 := TRUE;
ELSE
    _stAxis.stStatus.bCoupledGear3 := FALSE;
END_IF

IF _stAxis.Axis.Status.Coupled AND _stAxis.Axis.PlcToNc.GearRatio4 <> 0 AND _stAxis.stConfig.astMultiMasterAxisLatched[4].nIndex <> 0 THEN
    GVL.astAxes[_stAxis.stConfig.astMultiMasterAxisLatched[4].nIndex].stConfig.afMultiSlaveAxisRatio[GVL.iAxis] := _stAxis.Axis.PlcToNc.GearRatio4;
    _stAxis.stStatus.bCoupledGear4 := TRUE;
ELSE
    _stAxis.stStatus.bCoupledGear4 := FALSE;
END_IF
END_METHOD

METHOD mStatus_NewCommand : BOOL
VAR
    i: UINT;
END_VAR

fbExecuteRTrig(CLK := _stAxis.stControl.bExecute);
IF fbExecuteRTrig.Q THEN
    _stAxis.stStatus.bDone := FALSE;
    _stAxis.stStatus.bCommandAborted := FALSE;

    //On a new motion command, clear the errorID
    CASE _stAxis.stControl.eCommand OF
            E_MotionFunctions.eMoveAbsolute,
            E_MotionFunctions.eMoveRelative,
            E_MotionFunctions.eMoveVelocity,
            E_MotionFunctions.eMoveModulo,
            E_MotionFunctions.eGearInMultiMaster,
            E_MotionFunctions.eGearOut,
            E_MotionFunctions.eHome :
                _stAxis.stStatus.nErrorID := 0;
            E_MotionFunctions.eWriteParameter,
            E_MotionFunctions.eReadParameter :
            // Nothing
    END_CASE
END_IF
END_METHOD

METHOD Run : BOOL

mStatus_AxisStatus();
mParameters_ReadNc();
mParameters_Init();
stMcStatusReadParameter := mParameters_ReadParameter();
stMcStatusWriteParameter := mParameters_WriteParameter();

mControl_LimitHitTimer();
mControl_LimitLinking();
stMcStatusPower := mControl_Power();

stMcStatusHalt := mMove_Halt();
stMcStatusStop := mMove_Stop();
stMcStatusReset := mControl_Reset();

stMcStatusMoveAbsolute := mMove_MoveAbsolute();
stMcStatusMoveRelative := mMove_MoveRelative();
stMcStatusMoveModulo := mMove_MoveModulo();
stMcStatusMoveVelocity := mMove_MoveVelocity();

stMcStatusGearInMultiMaster := mControl_GearInMultiMaster();
stMcStatusGearOut := mControl_GearOut();

stMcStatusHome := mControl_Home();

mStatus_NewCommand();
mStatus_Done();
mStatus_Error();
mStatus_InVelocity();
mStatus_CommandAborted();
_stAxis.stStatus.bBusy := mStatus_Busy();

EndOfCycle();
END_METHOD

PROPERTY stAxis : REFERENCE TO ST_AxisStruct
GET
stAxis REF= _stAxis;
END_GET
SET
_stAxis REF= stAxis;
END_SET
END_PROPERTY

END_FUNCTION_BLOCK

// ---- tc_mca_std_lib/POUs/Motion/Homing/FB_Homing.TcPOU
FUNCTION_BLOCK FB_Homing
VAR_IN_OUT
    Axis: Axis_Ref;
END_VAR
VAR_INPUT
    bExecute: BOOL;
    bLimitFwd: BOOL;
    bLimitBwd: BOOL;
    bHomeSensor: BOOL;
    eHomeSeq: E_HomingRoutines;
    fHomePosition: LREAL;
    fHomeFinishDistance: LREAL;
    stConfig: ST_AxisConfig;
END_VAR
VAR_OUTPUT
    bDone : BOOL;
    bBusy: BOOL;
    bCommandAborted: BOOL;
    bError: BOOL;
    nErrorId: UDINT;
END_VAR
VAR
    //Beckhoff homing function blocks
    fbStepLimitSwitchPreparation: MC_StepLimitSwitchDetection;
    fbStepLimitSwitchDetection: MC_StepLimitSwitchDetection;
    fbStepAbsoluteSwitchDetection: MC_StepAbsoluteSwitchDetection;
    fbStepReferencePulseDetection: MC_StepReferencePulseDetection;
    fbStepBlockLagDetection: MC_StepBlockLagBasedDetection;
    fbHomeDirect: MC_HomeDirect;
    fbSetPos: MC_SetPosition;
    fbFinishHoming: MC_FinishHoming;
    fbAbortHoming: MC_AbortHoming;
    //Hardware Signals
    ePreparationLimitSwitchMode: MC_Switch_Mode := mcRisingEdge;
    stLimitSwitchSignal: MC_Ref_Signal_Ref;
    stRefSwitchSignal: MC_Ref_Signal_Ref;
    stEncPulseSignal: MC_Ref_Signal_Ref;
    //Homing parameters
    stPreparationDirection: MC_Home_Direction;
    stDetectDirection: MC_Home_Direction;
    stHomingParameter: MC_HomingParameter;
    stOptions: ST_Home_Options4;
    stOptions3: ST_Home_Options3;
    fbVelocityToCam: MC_ReadParameter;
    fVelocityToCam: LREAL;
    fbVelocityFromCam: MC_ReadParameter;
    fVelocityFromCam: LREAL;
    //State machine
    fbExecute: R_TRIG;
    bViaLimitSwitch: BOOL;
    eHomingState: (eWaitForRequest := 0, ePreparation := 1, eDetection := 2, eSetPos := 3, eFinishHoming := 4, eAbortHoming := 20);
    iErrorId: UDINT;
    bDetectionFB_Execute: BOOL;
    bDetectionFB_Done: BOOL;
    bDetectionFB_Busy: BOOL;
    bDetectionFB_CommandAborted: BOOL;
    bDetectionFB_Error: BOOL;
    nDetectionFB_ErrorID: UDINT;
    fRecordedPosition: LREAL;
    fRecordedPositionLatched: LREAL;
END_VAR


//Hardware signals
stLimitSwitchSignal.SignalSource := SignalSource_Default;
stLimitSwitchSignal.TouchProbe := PlcEvent;
stRefSwitchSignal.SignalSource := SignalSource_Default;
stRefSwitchSignal.TouchProbe := PlcEvent;
stRefSwitchSignal.Level := bHomeSensor;
stEncPulseSignal.SignalSource := SignalSource_ZeroPulse;
stEncPulseSignal.TouchProbe := TouchProbe1;

//Constantly read the NC for homing velocities so they are available when a homing is executed
fbVelocityToCam(
    Axis := Axis,
    Enable := TRUE,
    ParameterNumber := E_AxisParameters.AxisVelocityToCam,
    ReadMode := READMODE_CYCLIC);

fbVelocityFromCam(
    Axis := Axis,
    Enable := TRUE,
    ParameterNumber := E_AxisParameters.AxisVelocityFromCam,
    ReadMode := READMODE_CYCLIC);

    //Only write velocity if the function block has not errored
IF NOT fbVelocityToCam.Error THEN
    fVelocityToCam := fbVelocityToCam.Value;
END_IF

IF NOT fbVelocityFromCam.Error THEN
    fVelocityFromCam := fbVelocityFromCam.Value;
END_IF

    //Feeds function block errors through
IF fbVelocityToCam.Error THEN
    bError := TRUE;
    nErrorID := fbVelocityToCam.ErrorID;

ELSIF fbVelocityFromCam.Error THEN
    bError := TRUE;
    nErrorID := fbVelocityFromCam.ErrorID;
END_IF

//Common function blocks used for all routines
stOptions.DisableDriveAccess := stConfig.stHomingConfig.bDisableDriveAccess;
stOptions.EnableLagErrorDetection := stConfig.stHomingConfig.bEnableLagErrorDetection;

//For StepBlockLagDetection
stOptions3.DisableDriveAccess := stConfig.stHomingConfig.bDisableDriveAccess;
stOptions3.InstantLagReduction := stConfig.stHomingConfig.bInstantLagReduction;

fbStepLimitSwitchPreparation.Options.DisableDriveAccess := stOptions.DisableDriveAccess;
fbStepLimitSwitchPreparation(
    Axis := Axis,
    Parameter := stHomingParameter,
    Direction := stPreparationDirection,
    LimitSwitchMode:= ePreparationLimitSwitchMode,
    LimitSwitchSignal:= stLimitSwitchSignal,
    Velocity := fVelocityToCam);

fbSetPos(
    Axis := Axis,
    Position := Axis.NcToPlc.ActPos - fRecordedPositionLatched + fHomePosition);

fbFinishHoming.Options.DisableDriveAccess := stOptions.DisableDriveAccess;
fbFinishHoming(
    Axis := Axis,
    Parameter := stHomingParameter,
    Velocity := fVelocityFromCam);

fbAbortHoming.Options.DisableDriveAccess := stOptions.DisableDriveAccess;
fbAbortHoming(
    Axis := Axis,
    Parameter := stHomingParameter);

//ACTs contain function blocks custom to each individual routine for the detection stage
CASE eHomeSeq OF
    E_HomingRoutines.eHomeToLimit_Bwd,
    E_HomingRoutines.eHomeToLimit_Fwd:
        actHomeToLimit();

    E_HomingRoutines.eHomeToRef_Bwd,
    E_HomingRoutines.eHomeToRef_Fwd:
        actHomeToRef();

    E_HomingRoutines.eHomeToEncPulse_Bwd,
    E_HomingRoutines.eHomeToEncPulse_Fwd,
    E_HomingRoutines.eHomeToEncPulse_viaBwdLimit,
    E_HomingRoutines.eHomeToEncPulse_viaFwdLimit:
        actHomeToEncPulse();

    E_HomingRoutines.eHomeToBlock_Bwd,
    E_HomingRoutines.eHomeToBlock_Fwd:
        actHomeToBlock();

    E_HomingRoutines.eHomeDirect:
        actHomeDirect();
END_CASE


//State machine
fbExecute(CLK:= bExecute);
CASE eHomingState OF

    eWaitForRequest:
        IF NOT bExecute THEN
            bBusy := FALSE;
            bDone := FALSE;
            bCommandAborted := FALSE;
            bError := FALSE;
            nErrorID := 0;
            iErrorID := 0;

            fbStepLimitSwitchPreparation.Execute := FALSE;
            fbStepLimitSwitchDetection.Execute := FALSE;
            fbStepAbsoluteSwitchDetection.Execute := FALSE;
            fbStepReferencePulseDetection.Execute := FALSE;
            fbStepBlockLagDetection.Execute := FALSE;
            fbHomeDirect.Execute := FALSE;
            fbSetPos.Execute := FALSE;
            fbFinishHoming.Execute := FALSE;
            fbAbortHoming.Execute := FALSE;
        END_IF

        IF fbExecute.Q AND NOT(eHomeSeq = E_HomingRoutines.eNoHoming)THEN
            bBusy:= TRUE;
            eHomingState:= ePreparation;
        END_IF


    ePreparation: //If bViaLimitSwitch is set TRUE then go first to a limit otherwise skip this step
        IF bViaLimitSwitch THEN
            fbStepLimitSwitchPreparation.Execute := TRUE;
        ELSE
            eHomingState := eDetection;
        END_IF

        IF NOT fbStepLimitSwitchPreparation.Busy AND fbStepLimitSwitchPreparation.Done THEN
            fbStepLimitSwitchPreparation.Execute := FALSE;
            eHomingState := eDetection;
        ELSIF NOT fbStepLimitSwitchPreparation.Busy AND (fbStepLimitSwitchPreparation.Error OR fbStepLimitSwitchPreparation.CommandAborted) THEN
            iErrorID := fbStepLimitSwitchPreparation.ErrorID;
            fbStepLimitSwitchPreparation.Execute := FALSE;
            eHomingState := eAbortHoming;
        END_IF


    eDetection: //Use bDetectionFB_<BOOL Variables> to interact with different detection FBs located in ACTs
        bDetectionFB_Execute := TRUE;

        IF NOT bDetectionFB_Busy AND bDetectionFB_Done THEN
            bDetectionFB_Execute := FALSE;
            fRecordedPositionLatched := fRecordedPosition;
            IF eHomeSeq = E_HomingRoutines.eHomeDirect THEN
                bBusy := fbHomeDirect.Busy;
                bDone := fbHomeDirect.Done;
                bCommandAborted := fbHomeDirect.CommandAborted;
                bError := fbHomeDirect.Error;
                nErrorId := fbHomeDirect.ErrorID;
                eHomingState := eWaitForRequest;
            ELSE
                eHomingState := eSetPos;
            END_IF
        ELSIF NOT bDetectionFB_Busy AND (bDetectionFB_Error OR bDetectionFB_CommandAborted) THEN
            iErrorID := nDetectionFB_ErrorID;
            bDetectionFB_Execute := FALSE;
            eHomingState := eAbortHoming;
        END_IF


    eSetPos:
        fbSetPos.Execute := TRUE;

        fbSetPos.Options.ClearPositionLag := TRUE;
        IF NOT fbSetPos.Busy AND fbSetPos.Done THEN
            fbSetPos.Execute := FALSE;
            eHomingState := eFinishHoming;
        ELSIF NOT fbSetPos.Busy AND fbSetPos.Error THEN
            iErrorID := fbSetPos.ErrorID;
            fbSetPos.Execute := FALSE;
            eHomingState := eAbortHoming;
        END_IF


    eFinishHoming:
        fbFinishHoming.Execute := TRUE;

        IF NOT fbFinishHoming.Busy AND fbFinishHoming.Done THEN
            bBusy := FALSE;
            bDone := TRUE;
            fbFinishHoming.Execute := FALSE;
            eHomingState := eWaitForRequest;
        ELSIF NOT fbFinishHoming.Busy AND (fbFinishHoming.Error OR fbFinishHoming.CommandAborted) THEN
            iErrorID := fbFinishHoming.ErrorID;
            fbFinishHoming.Execute := FALSE;
            eHomingState := eAbortHoming;
        END_IF


    eAbortHoming:
        fbAbortHoming.Execute := TRUE;

        IF NOT fbAbortHoming.Busy AND fbAbortHoming.Done THEN
            bBusy := FALSE;
            IF iErrorId <> 0 THEN
                bError := TRUE;
                nErrorId := iErrorId;
            ELSE
                bCommandAborted := TRUE;
            END_IF
            fbAbortHoming.Execute := FALSE;
            eHomingState := eWaitForRequest;
        ELSIF NOT fbAbortHoming.Busy AND fbAbortHoming.Error THEN
            bBusy := FALSE;
            bError := TRUE;
            nErrorID := fbAbortHoming.ErrorID;
            fbAbortHoming.Execute := FALSE;
            eHomingState := eWaitForRequest;
        END_IF

END_CASE

ACTION actHomeDirect:

bViaLimitSwitch := FALSE;

fbHomeDirect(
    Axis := Axis,
    Parameter := stHomingParameter,
    Execute := bDetectionFB_Execute,
    SetPosition := fHomePosition,
    Done => bDetectionFB_Done,
    Busy => bDetectionFB_Busy,
    CommandAborted => bDetectionFB_CommandAborted,
    Error => bDetectionFB_Error,
    ErrorID => nDetectionFB_ErrorID);
END_ACTION

ACTION actHomeToBlock:
CASE eHomeSeq OF
    E_HomingRoutines.eHomeToBlock_Bwd:
        stDetectDirection:= mcNegativeDirection;
        fbFinishHoming.Distance := fHomeFinishDistance;
    E_HomingRoutines.eHomeToBlock_Fwd:
        stDetectDirection:= mcPositiveDirection;
        fbFinishHoming.Distance := -fHomeFinishDistance;
END_CASE

bViaLimitSwitch:=FALSE;

fbStepBlockLagDetection(
    Axis := Axis,
    Execute := bDetectionFB_Execute,
    Parameter := stHomingParameter,
    Direction := stDetectDirection,
    Velocity := fVelocityFromCam, //Maximum travel velocity (>0).
    DetectionVelocityLimit := stConfig.stHomingConfig.fDetectionVelocityLimit, //Velocity that must be fallen below for the time DetectionVelocityTime in order to detect driving against the fixed stop.
    DetectionVelocityTime := stConfig.stHomingConfig.tDetectionVelocityTime, //Time for detecting the velocity undershoot when driving against the fixed stop.
    TimeLimit :=  stConfig.stHomingConfig.tTimeLimit, //Exceeding this time leads to the search procedure being aborted.
    DistanceLimit := stConfig.stHomingConfig.fDistanceLimit, //Exceeding this distance in relation to the start position leads to the search procedure being aborted.
    TorqueLimit := stConfig.stHomingConfig.fTorqueLimit, //The motor torque is limited to this value (percentage of configured channel peak torque), in relation to the weight counterbalance that is possibly parameterized in the drive, in order to avoid mechanical damage.
    LagLimit := stConfig.stHomingConfig.fLagLimit, //Position lag value which, if exceeded, leads to detection of driving against the fixed stop.
    Options := stOptions3,
    Done => bDetectionFB_Done,
    Busy => bDetectionFB_Busy,
    CommandAborted => bDetectionFB_CommandAborted,
    Error => bDetectionFB_Error,
    ErrorID => nDetectionFB_ErrorID,
    RecordedPosition => fRecordedPosition);
END_ACTION

ACTION actHomeToEncPulse:

CASE eHomeSeq OF
    E_HomingRoutines.eHomeToEncPulse_Bwd:
        stDetectDirection := mcNegativeDirection;
        fbFinishHoming.Distance := fHomeFinishDistance;
        bViaLimitSwitch := FALSE;
    E_HomingRoutines.eHomeToEncPulse_Fwd:
        stDetectDirection := mcPositiveDirection;
        fbFinishHoming.Distance := -fHomeFinishDistance;
        bViaLimitSwitch := FALSE;
    E_HomingRoutines.eHomeToEncPulse_viaBwdLimit:
        stDetectDirection := mcPositiveDirection;
        fbFinishHoming.Distance := fHomeFinishDistance;
        stPreparationDirection := mcNegativeDirection;
        stLimitSwitchSignal.Level := NOT(bLimitBwd);
        bViaLimitSwitch := TRUE;
    E_HomingRoutines.eHomeToEncPulse_viaFwdLimit:
        stDetectDirection := mcNegativeDirection;
        fbFinishHoming.Distance := -fHomeFinishDistance;
        stPreparationDirection := mcPositiveDirection;
        stLimitSwitchSignal.Level := NOT(bLimitFwd);
        bViaLimitSwitch := TRUE;
END_CASE

fbStepReferencePulseDetection.Options.DisableDriveAccess:= stOptions.DisableDriveAccess;
fbStepReferencePulseDetection(
    Axis := Axis,
    Execute := bDetectionFB_Execute,
    Parameter := stHomingParameter,
    Direction := stDetectDirection,
    ReferenceSignal := stEncPulseSignal,
    Velocity := fVelocityFromCam,
    Options := stOptions,
    Done => bDetectionFB_Done,
    Busy => bDetectionFB_Busy,
    CommandAborted => bDetectionFB_CommandAborted,
    Error => bDetectionFB_Error,
    ErrorID => nDetectionFB_ErrorID,
    RecordedPosition => fRecordedPosition);
END_ACTION

ACTION actHomeToLimit:

CASE eHomeSeq OF
    E_HomingRoutines.eHomeToLimit_Bwd:
        stLimitSwitchSignal.Level := NOT(bLimitBwd);
        stDetectDirection:= mcNegativeDirection;
        fbFinishHoming.Distance := fHomeFinishDistance;
    E_HomingRoutines.eHomeToLimit_Fwd:
        stLimitSwitchSignal.Level := NOT(bLimitFwd);
        stDetectDirection:= mcPositiveDirection;
        fbFinishHoming.Distance := -fHomeFinishDistance;
END_CASE
bViaLimitSwitch:=FALSE;

fbStepLimitSwitchDetection.Options.DisableDriveAccess:= stOptions.DisableDriveAccess;
fbStepLimitSwitchDetection(
    Axis := Axis,
    Execute := bDetectionFB_Execute,
    Parameter := stHomingParameter,
    Direction := stDetectDirection,
    LimitSwitchMode := stConfig.stHomingConfig.eLimitSwitchMode,
    LimitSwitchSignal := stLimitSwitchSignal,
    Velocity := fVelocityFromCam,
    Options := stOptions,
    Done => bDetectionFB_Done,
    Busy => bDetectionFB_Busy,
    CommandAborted => bDetectionFB_CommandAborted,
    Error => bDetectionFB_Error,
    ErrorID => nDetectionFB_ErrorID,
    RecordedPosition => fRecordedPosition);
END_ACTION

ACTION actHomeToRef:

